METHOD FB_init : BOOL
VAR_INPUT
  /// if TRUE, the retain variables are initialized (warm start / cold start)
  bInitRetains : BOOL; 
  /// if TRUE, the instance afterwards gets moved into the copy code (online change)
  bInCopyCode  : BOOL;  
END_VAR
                  MyType := 'MC_MoveDirectOffsetFB';

ExecMode     := ExecutionMode.SEQUENCE_PRIMARY;
Priority     := PriorityLevel.NORMAL;
AbortingMode := AbortingModeEnum.BUFFER;  
SequenceFlag := SequenceFlagEnum.PRIMARY_SEQUENCE;  

                
END_METHOD

METHOD PROTECTED OnApplyOutCmd
VAR_INPUT
  /// Command message state
  State : CmdMessageState;
END_VAR
                  IF ( State = CmdMessageState.EMPTY ) 
THEN
  // Reset command outputs
  SysDepMemSet(pDest := ADR(OutCmd), Value := 0, DataLen := SIZEOF(OutCmd));         
END_IF

IF (( State = CmdMessageState.ACTIVE ) OR
    ( State = CmdMessageState.DONE   ))
THEN
  // Update results
  OutCmd.Progress          :=  PERCENT_UINT_TO_REAL( Value := _response.Progress, IsOptional := TRUE);
  OutCmd.FollowID          := _response.OriginID;
  OutCmd.RemainingDistance := _response.RemainingDistance;
END_IF
                
END_METHOD

METHOD PROTECTED OnExecRun : DINT
VAR_IN_OUT
  /// Robot assignment of function
  AxesGroup : AxesGroup; 
END_VAR
                  // call base implementation
SUPER^.OnExecRun(AxesGroup := AxesGroup);

CASE _stepCmd OF
  
  00:  IF ( _execute_R.Q ) AND ( NOT Error)  
       THEN
         // Check function is supported and parameter are valid ?
         IF (( CheckFunctionSupported( AxesGroup := AxesGroup )) AND
             ( CheckParameterValid   ( AxesGroup := AxesGroup )))      
         THEN
           // set busy flag
           Busy := TRUE;
           // Reset command outputs
           SysDepMemSet(pDest := ADR(OutCmd), Value := 0, DataLen := SIZEOF(OutCmd));         
           // apply command parameter
          _parCmd := ParCmd;
           // init parameter sequence
          _command.ParSeq := 1;
           // create command data
           CommandData := CreateCommandPayload(AxesGroup := AxesGroup);
           // Add command to active command register
          _uniqueID := AxesGroup.Acyclic.ActiveCommandRegister.AddCmd( pCommandFB := ADR(THIS^ ));     
           // set timeout
           SetTimeout(PT := _timeoutCmd, rTimer := _timerCmd);
           // inc step counter
          _stepCmd := _stepCmd + 1;
         END_IF 
       END_IF
     

  01:  // Wait for responce received
       IF ( _responseReceived )
       THEN
         // reset response received flag
        _responseReceived := FALSE;
         // update state flags
         OnUpdateStateFlags(_response.State);
         // update state flags
         OnApplyOutCmd(_response.State);
        
         // Done, Aborted or Error ?
         IF (_response.State >= CmdMessageState.DONE )
         THEN
           // set timeout
           SetTimeout(PT := _timeoutCmd, rTimer := _timerCmd);
           // inc step counter
          _stepCmd := _stepCmd + 1; 
         END_IF
       END_IF


  02: IF ( NOT Execute)
      THEN
        Reset();  
      END_IF     
ELSE
  // invalid step
  SetError( ErrorID := RobotLibraryErrorIdEnum.ERR_INVALID_STEP, Overwrite := TRUE );
END_CASE


// Reset FB
IF ( NOT Execute )
THEN
  Reset(); 
END_IF
                
END_METHOD

METHOD PROTECTED OnUpdateStateFlags
VAR_INPUT
  /// Command message state
  State : CmdMessageState;
END_VAR
                  // Reset State flags
Active             := FALSE;
CommandAborted     := FALSE;
CommandInterrupted := FALSE;
Done               := FALSE;

CASE State OF

  // No operation or process is active
  CmdMessageState.EMPTY               :;
  // Created but not yet started
  CmdMessageState.CREATED             :;
  // Buffered and awaiting execution
  CmdMessageState.BUFFERED            : CommandBuffered    := TRUE;
  // Buffered in planner for future execution
  CmdMessageState.BUFFERED_IN_PLANNER : CommandBuffered    := TRUE;
  // Currently active and in progress
  CmdMessageState.ACTIVE              : Active             := TRUE; 
  // Interrupted and awaiting continuation
  CmdMessageState.INTERRUPTED         : CommandInterrupted := TRUE;  
  // Requested for abort
  CmdMessageState.ABORT_REQUEST       :;
  // Successfully completed
  CmdMessageState.DONE                : Done               := TRUE;
                                        Busy               := FALSE;
  // Aborted before completion
  CmdMessageState.ABORTED             : CommandAborted     := TRUE;
                                        Busy               := FALSE;
  // Encountered an error during execution
  CmdMessageState.ERROR               : Error              := TRUE;
                                        Busy               := FALSE;
END_CASE
                
END_METHOD

METHOD INTERNAL ParseResponsePayload : DINT
VAR_INPUT
  /// Response data
  ResponseData : RobotLibraryResponseDataFB;
  /// Timestamp
  Timestamp    : SystemTime;  
END_VAR
VAR
  /// Parameter count
 _parameterCnt : DINT;
END_VAR
// Table 6-354: Received CMD payload (RC to PLC) of "MoveDirectOffset"
// --------------------------
// Header
// --------------------------
// Byte 00 : USINT   - ParSeq | State     
// Byte 01 : SINT    - AlarmMessageSeverity    
// Byte 02 : UINT    - AlarmMessageCode HB
// Byte 03 :         - AlarmMessageCode LB
// --------------------------
// Datablock
// --------------------------
// Byte 04 : USINT      - InvocationCounter
// Byte 05 : SINT       - Reserved
// Byte 06 : INT        - OriginID HW HB
// Byte 07 :            - OriginID HW LB
// Byte 08 : UINT       - Progress HW HB
// Byte 09 :            - Progress HW LB
// Byte 10 : REAL       - RemainingDistance HW HB
// Byte 11 :            - RemainingDistance HW LB
// Byte 12 :            - RemainingDistance LW HB
// Byte 13 :            - RemainingDistance LW LB
                  // call base implementation to parse the header from payload buffer
ResponseData.PayloadPtr := SUPER^.ParseResponsePayload(ResponseData := ResponseData, Timestamp := Timestamp);

// copy parsed header to response
_response.ParSeq               := _rspHeader.ParSeq;
_response.State                := _rspHeader.State;
_response.AlarmMessageSeverity := _rspHeader.AlarmMessageSeverity;
_response.AlarmMessageCode     := _rspHeader.AlarmMessageCode;


// Check payload remaining ? 
IF ( ResponseData.IsPayloadRemaining)
THEN
  // Get Response.InvocationCounter
 _response.InvocationCounter := ResponseData.GetUsint();
  // inc parameter counter
 _parameterCnt := _parameterCnt + 1;
END_IF

// Check payload remaining ? 
IF ( ResponseData.IsPayloadRemaining)
THEN
  // Get Response.Reserve
 _response.Reserve := ResponseData.GetSint();
  // inc parameter counter
 _parameterCnt := _parameterCnt + 1;
END_IF


// Check payload remaining ? 
IF ( ResponseData.IsPayloadRemaining)
THEN
  // Get Response.OriginID
 _response.OriginID := ResponseData.GetInt();
  // inc parameter counter
 _parameterCnt := _parameterCnt + 1;
END_IF


// Check payload remaining ? 
IF ( ResponseData.IsPayloadRemaining)
THEN
  // Get Response.Progress
 _response.Progress := ResponseData.GetUint();
  // inc parameter counter
 _parameterCnt := _parameterCnt + 1;
END_IF


// Check payload remaining ? 
IF ( ResponseData.IsPayloadRemaining)
THEN
  // Get Response.RemainingDistance
 _response.RemainingDistance := ResponseData.GetReal();
  // inc parameter counter
 _parameterCnt := _parameterCnt + 1;
END_IF
 
 
// Create logging
ParseResponsePayloadLog(ResponseData := ResponseData, Timestamp := Timestamp, ParameterCnt := _parameterCnt);
                
END_METHOD

METHOD INTERNAL ParseResponsePayloadLog
VAR_INPUT
  /// Response data
  ResponseData : RobotLibraryResponseDataFB;
  /// Timestamp
  Timestamp    : SystemTime;  
  /// Parameter count
  ParameterCnt : DINT;
END_VAR
                  // Create log entry for Parameter start
CreateLogMessagePara1 ( Timestamp   := Timestamp,
                        MessageType := MessageType.CMD,
                        Severity    := Severity.DEBUG,
                        MessageCode := 0,
                        MessageText := '{1} parameter(s) to parse from the response data:',
                        Para1       := DINT_TO_STRING(ParameterCnt));
                        

// Return if no parameter is remaining...
IF ( ParameterCnt = 0 ) THEN RETURN; END_IF
// dec remaining parameter(s)                        
ParameterCnt := ParameterCnt - 1;
// Create log entry for InvocationCounter
CreateLogMessagePara1 ( Timestamp   := Timestamp,
                        MessageType := MessageType.CMD,
                        Severity    := Severity.DEBUG,
                        MessageCode := 0,
                        MessageText := 'Response.InvocationCounter = {1}',
                        Para1       :=  USINT_TO_STRING(_response.InvocationCounter));


// Return if no parameter is remaining...
IF ( ParameterCnt = 0 ) THEN RETURN; END_IF
// dec remaining parameter(s)                        
ParameterCnt := ParameterCnt - 1;
// Create log entry for Reserve
CreateLogMessagePara1 ( Timestamp   := Timestamp,
                        MessageType := MessageType.CMD,
                        Severity    := Severity.DEBUG,
                        MessageCode := 0,
                        MessageText := 'Response.Reserve = {1}',
                        Para1       :=  SINT_TO_STRING(_response.Reserve));


// Return if no parameter is remaining...
IF ( ParameterCnt = 0 ) THEN RETURN; END_IF
// dec remaining parameter(s)                        
ParameterCnt := ParameterCnt - 1;
// Create log entry for OriginID
CreateLogMessagePara1 ( Timestamp   := Timestamp,
                        MessageType := MessageType.CMD,
                        Severity    := Severity.DEBUG,
                        MessageCode := 0,
                        MessageText := 'Response.OriginID = {1}',
                        Para1       :=  INT_TO_STRING(_response.OriginID));


// Return if no parameter is remaining...
IF ( ParameterCnt = 0 ) THEN RETURN; END_IF
// dec remaining parameter(s)                        
ParameterCnt := ParameterCnt - 1;
// Create log entry for Progress
CreateLogMessagePara1 ( Timestamp   := Timestamp,
                        MessageType := MessageType.CMD,
                        Severity    := Severity.DEBUG,
                        MessageCode := 0,
                        MessageText := 'Response.Progress = {1}',
                        Para1       :=  UINT_TO_STRING(_response.Progress));


// Return if no parameter is remaining...
IF ( ParameterCnt = 0 ) THEN RETURN; END_IF
// dec remaining parameter(s)                        
ParameterCnt := ParameterCnt - 1;
// Create log entry for RemainingDistance
CreateLogMessagePara1 ( Timestamp   := Timestamp,
                        MessageType := MessageType.CMD,
                        Severity    := Severity.DEBUG,
                        MessageCode := 0,
                        MessageText := 'Response.RemainingDistance = {1}',
                        Para1       :=  REAL_TO_STRING(_response.RemainingDistance));
                
END_METHOD

METHOD PROTECTED Reset : DINT
VAR_INPUT
END_VAR
                  Reset := SUPER^.Reset();

Done               := FALSE;
Busy               := FALSE;
Active             := FALSE;
CommandBuffered    := FALSE;
CommandAborted     := FALSE;
CommandInterrupted := FALSE;

                
END_METHOD
END_FUNCTION_BLOCK

/// Move Joints relative to relative cartesian position (Relative cartesian PTP) (Joint interpolated movement)
FUNCTION_BLOCK MC_MoveDirectRelativeFB EXTENDS RobotLibraryBaseExecuteFB
// ------------------------------------------------------------------------- 
//  SRCI Robot Library                                                
// ------------------------------------------------------------------------- 
//                                                                           
//  Object:      MoveDirectRelativeFB                                       
//  Author:      Thorsten Brach                                                
//  Date:        2024-06-01
//
//  Description:                                              
//   
//                                                                           
//  Copyright: 
//    (C) 2024 Thorsten Brach. All rights reserved                                                                                                                                            
//             Licensed under the MIT License.
//                                                                           
//  Disclaimer:                                                                           
//    This project is provided without any guarantee and can be used for   
//    private and commercial purposes. Any use is at the user’s 
//    own risk and responsibility.
//
// -------------------------------------------------------------------------
VAR_INPUT
  /// Parameter which determines the behavior towards the previously sent and still active or buffered commands
  AbortingMode       : AbortingMode;
  /// Defines the target sequence in which the command will be executed
  SequenceFlag       : SequenceFlag;
  /// command parameter
  ParCmd             : MoveDirectRelativeParCmd;       
END_VAR

VAR_OUTPUT
  /// Command is transferred and confirmed by the RC
  CommandBuffered    : BOOL;
  /// The command takes control of the motion of the according axis group
  Active             : BOOL;
  /// The command was aborted by another command.
  CommandAborted     : BOOL;
  /// TRUE, while command is interrupted during execution and can be continued
  CommandInterrupted : BOOL;
  /// command outputs
  OutCmd             : MoveDirectRelativeOutCmd;       
END_VAR



VAR
  /// internal copy of command parameter 
 _parCmd             : MoveDirectRelativeParCmd;
  /// command data to send
 _command            : MoveDirectRelativeSendData;
  /// response data received
 _response           : MoveDirectRelativeRecvData;      
END_VAR

            SUPER^(AxesGroup := AxesGroup);
          

METHOD INTERNAL CheckAddParameter : BOOL
VAR_INPUT
  /// Payload pointer
  PayloadPtr : UDINT;
END_VAR
VAR
  /// Payload as byte array
  Payload    : ARRAY [1..SIZEOF(_command)] OF BYTE;
  /// Null Byte array 
  Null       : ARRAY [1..SIZEOF(_command)] OF BYTE;
  /// Data length to compare
  DataLen    : UDINT;
END_VAR
                  // Payload pointer must be decreased by one byte, because ADR(Payload) is already one byte !
PayloadPtr := LIMIT (0, PayloadPtr - 1, SIZEOF(Payload) -1);
// Convert command struct to payload array
SysDepMemCpy( pDest := ADR(Payload), pSrc := ADR(_command), DataLen := SIZEOF(_command));
// Calculate the data length to compare - at least one byte must be compared !
DataLen := LIMIT(1, SIZEOF(Payload) - PayloadPtr, SIZEOF(Payload)); 
// Compare Payload-Array with Null-Byte-Array
CheckAddParameter := SysDepMemCmp( pData1 := ADR(Payload) + PayloadPtr , pData2 := ADR(Null), DataLen := DataLen) <>  RobotLibraryConstants.OK ;
                
END_METHOD

METHOD PROTECTED CheckFunctionSupported : BOOL
VAR_IN_OUT
  /// Robot assignment of function
  AxesGroup : AxesGroup; 
END_VAR
                  CheckFunctionSupported := AxesGroup.State.RobotData.RCSupportedFunctions.MoveDirectRelative;

IF ( NOT CheckFunctionSupported )
THEN
  // call base implementation for set error and create log entry
  SUPER^.CheckFunctionSupported(AxesGroup := AxesGroup);
END_IF
                
END_METHOD

METHOD PROTECTED CheckParameterChanged : BOOL
VAR_IN_OUT
  /// Robot assignment of function
  AxesGroup    : AxesGroup; 
END_VAR
                  // Check ParCmd Size is > 0, because MemCmp does not work correctly with size = 0
IF (SIZEOF(ParCmd) = 0) OR (_stepCmd = 0)
THEN 
  RETURN;
END_IF

// compare memory 
_parameterChanged := ( SysDepMemCmp(pData1 := ADR(ParCmd), pData2 := ADR(_parCmd), DataLen := SIZEOF(ParCmd)) <> RobotLibraryConstants.OK );

// check parameter valid ?
_parameterValid   := CheckParameterValid( AxesGroup := AxesGroup );

IF ((  _parameterChanged        )  AND 
    (  _parameterValid          )) OR
    (  _parameterUpdateInternal )  
THEN  
  // Create log entry for parameter changed event
  CreateLogMessagePara1 ( Timestamp   := AxesGroup.State.SystemTime,
                          MessageType := MessageType.CMD,
                          Severity    := Severity.DEBUG,
                          MessageCode := 0,
                          MessageText := 'NotifyParameterChanged Event {1}',
                          Para1       :=  '' );

  // reset internal flag for send parameter update
 _parameterUpdateInternal := FALSE;
  // update internal copy of parameters 
 _parCmd := ParCmd;
  // inc parameter sequence
 _command.ParSeq := _command.ParSeq + 1;
  // update command data  
  CommandData := CreateCommandPayload(AxesGroup := AxesGroup); // ( Access via reference to rCommandFB in ACR )
  // notify active command register 
  AxesGroup.Acyclic.ActiveCommandRegister.NotifyParameterChanged := _uniqueID;
END_IF
                
END_METHOD

METHOD PROTECTED CheckParameterValid : BOOL
VAR_IN_OUT
  /// Robot assignment of function
  AxesGroup : AxesGroup; 
END_VAR
VAR
  /// internal index for loops
 _idx : DINT;
END_VAR
                  CheckParameterValid := TRUE;

// Check AbortingMode valid ? 
IF (( AbortingMode <> AbortingModeEnum.BUFFER ) AND
    ( AbortingMode <> AbortingModeEnum.ABORT  ))  
THEN
  // Parameter not valid
  CheckParameterValid := FALSE;
  // Set error
  SetError( ErrorID := RobotLibraryErrorIdEnum.ERR_ABORTINGMODE_INVALID, Overwrite := TRUE );
  // Create log entry
  CreateLogMessagePara1 ( Timestamp   := AxesGroup.State.SystemTime,
                          MessageType := MessageType.CMD,
                          Severity    := Severity.ERROR,
                          MessageCode := ErrorID,
                          MessageText := 'Invalid Parameter AbortingMode = {1}',
                          Para1       := ABORTING_MODE_TO_STRING(AbortingMode));
  RETURN;                          
END_IF


// Check SequenceFlag valid ? 
IF (( SequenceFlag <> SequenceFlagEnum.PRIMARY_SEQUENCE   ) AND
    ( SequenceFlag <> SequenceFlagEnum.SECONDARY_SEQUENCE ))
THEN
  // Parameter not valid
  CheckParameterValid := FALSE;
  // Set error
  SetError( ErrorID := RobotLibraryErrorIdEnum.ERR_SEQFLAG_NOT_ALLOWED, Overwrite := TRUE );
  // Create log entry
  CreateLogMessagePara1 ( Timestamp   := AxesGroup.State.SystemTime,
                          MessageType := MessageType.CMD,
                          Severity    := Severity.ERROR,
                          MessageCode := ErrorID,
                          MessageText := 'Invalid Parameter SequenceFlag = {1}',
                          Para1       := SEQUENCE_FLAG_TO_STRING(SequenceFlag));
  RETURN;                          
END_IF


// Check ParCmd.Distance.X valid ? 
IF ( SysDepIsValidReal(ParCmd.Distance.X) = FALSE ) 
THEN
  // Parameter not valid
  CheckParameterValid := FALSE;
  // Set error
  SetError( ErrorID := RobotLibraryErrorIdEnum.ERR_INVALID_PAR_CMD, Overwrite := TRUE );
  
  // Create log entry
  CreateLogMessagePara1 ( Timestamp   := AxesGroup.State.SystemTime,
                          MessageType := MessageType.CMD,
                          Severity    := Severity.ERROR,
                          MessageCode := ErrorID,
                          MessageText := 'Invalid Parameter ParCmd.Distance.X = {1}',
                          Para1       := VALID_REAL_TO_STRING(ParCmd.Distance.X));
  RETURN;                          
END_IF


// Check ParCmd.Distance.Y valid ? 
IF ( SysDepIsValidReal(ParCmd.Distance.Y) = FALSE ) 
THEN
  // Parameter not valid
  CheckParameterValid := FALSE;
  // Set error
  SetError( ErrorID := RobotLibraryErrorIdEnum.ERR_INVALID_PAR_CMD, Overwrite := TRUE );
  
  // Create log entry
  CreateLogMessagePara1 ( Timestamp   := AxesGroup.State.SystemTime,
                          MessageType := MessageType.CMD,
                          Severity    := Severity.ERROR,
                          MessageCode := ErrorID,
                          MessageText := 'Invalid Parameter ParCmd.Distance.Y = {1}',
                          Para1       := VALID_REAL_TO_STRING(ParCmd.Distance.Y));
  RETURN;                          
END_IF


// Check ParCmd.Distance.Z valid ? 
IF ( SysDepIsValidReal(ParCmd.Distance.Z) = FALSE ) 
THEN
  // Parameter not valid
  CheckParameterValid := FALSE;
  // Set error
  SetError( ErrorID := RobotLibraryErrorIdEnum.ERR_INVALID_PAR_CMD, Overwrite := TRUE );
  
  // Create log entry
  CreateLogMessagePara1 ( Timestamp   := AxesGroup.State.SystemTime,
                          MessageType := MessageType.CMD,
                          Severity    := Severity.ERROR,
                          MessageCode := ErrorID,
                          MessageText := 'Invalid Parameter ParCmd.Distance.Z = {1}',
                          Para1       := VALID_REAL_TO_STRING(ParCmd.Distance.Z));
  RETURN;                          
END_IF


// Check ParCmd.Distance.Rx valid ? 
IF ( SysDepIsValidReal(ParCmd.Distance.Rx) = FALSE ) 
THEN
  // Parameter not valid
  CheckParameterValid := FALSE;
  // Set error
  SetError( ErrorID := RobotLibraryErrorIdEnum.ERR_INVALID_PAR_CMD, Overwrite := TRUE );
  
  // Create log entry
  CreateLogMessagePara1 ( Timestamp   := AxesGroup.State.SystemTime,
                          MessageType := MessageType.CMD,
                          Severity    := Severity.ERROR,
                          MessageCode := ErrorID,
                          MessageText := 'Invalid Parameter ParCmd.Distance.Rx = {1}',
                          Para1       := VALID_REAL_TO_STRING(ParCmd.Distance.Rx));
  RETURN;                          
END_IF


// Check ParCmd.Distance.Ry valid ? 
IF ( SysDepIsValidReal(ParCmd.Distance.Ry) = FALSE ) 
THEN
  // Parameter not valid
  CheckParameterValid := FALSE;
  // Set error
  SetError( ErrorID := RobotLibraryErrorIdEnum.ERR_INVALID_PAR_CMD, Overwrite := TRUE );
  
  // Create log entry
  CreateLogMessagePara1 ( Timestamp   := AxesGroup.State.SystemTime,
                          MessageType := MessageType.CMD,
                          Severity    := Severity.ERROR,
                          MessageCode := ErrorID,
                          MessageText := 'Invalid Parameter ParCmd.Distance.Ry = {1}',
                          Para1       := VALID_REAL_TO_STRING(ParCmd.Distance.Ry));
  RETURN;                          
END_IF


// Check ParCmd.Distance.Rz valid ? 
IF ( SysDepIsValidReal(ParCmd.Distance.Rz) = FALSE ) 
THEN
  // Parameter not valid
  CheckParameterValid := FALSE;
  // Set error
  SetError( ErrorID := RobotLibraryErrorIdEnum.ERR_INVALID_PAR_CMD, Overwrite := TRUE );
  
  // Create log entry
  CreateLogMessagePara1 ( Timestamp   := AxesGroup.State.SystemTime,
                          MessageType := MessageType.CMD,
                          Severity    := Severity.ERROR,
                          MessageCode := ErrorID,
                          MessageText := 'Invalid Parameter ParCmd.Distance.Rz = {1}',
                          Para1       := VALID_REAL_TO_STRING(ParCmd.Distance.Rz));
  RETURN;                          
END_IF


// Check ParCmd.Distance.E1 valid ? 
IF ( SysDepIsValidReal(ParCmd.Distance.E1) = FALSE ) 
THEN
  // Parameter not valid
  CheckParameterValid := FALSE;
  // Set error
  SetError( ErrorID := RobotLibraryErrorIdEnum.ERR_INVALID_PAR_CMD, Overwrite := TRUE );
  
  // Create log entry
  CreateLogMessagePara1 ( Timestamp   := AxesGroup.State.SystemTime,
                          MessageType := MessageType.CMD,
                          Severity    := Severity.ERROR,
                          MessageCode := ErrorID,
                          MessageText := 'Invalid Parameter ParCmd.Distance.E1 = {1}',
                          Para1       := VALID_REAL_TO_STRING(ParCmd.Distance.E1));
  RETURN;                          
END_IF


// Check ParCmd.Distance.E2 valid ? 
IF ( SysDepIsValidReal(ParCmd.Distance.E2) = FALSE ) 
THEN
  // Parameter not valid
  CheckParameterValid := FALSE;
  // Set error
  SetError( ErrorID := RobotLibraryErrorIdEnum.ERR_INVALID_PAR_CMD, Overwrite := TRUE );
  
  // Create log entry
  CreateLogMessagePara1 ( Timestamp   := AxesGroup.State.SystemTime,
                          MessageType := MessageType.CMD,
                          Severity    := Severity.ERROR,
                          MessageCode := ErrorID,
                          MessageText := 'Invalid Parameter ParCmd.Distance.E2 = {1}',
                          Para1       := VALID_REAL_TO_STRING(ParCmd.Distance.E2));
  RETURN;                          
END_IF


// Check ParCmd.Distance.E3 valid ? 
IF ( SysDepIsValidReal(ParCmd.Distance.E3) = FALSE ) 
THEN
  // Parameter not valid
  CheckParameterValid := FALSE;
  // Set error
  SetError( ErrorID := RobotLibraryErrorIdEnum.ERR_INVALID_PAR_CMD, Overwrite := TRUE );
  
  // Create log entry
  CreateLogMessagePara1 ( Timestamp   := AxesGroup.State.SystemTime,
                          MessageType := MessageType.CMD,
                          Severity    := Severity.ERROR,
                          MessageCode := ErrorID,
                          MessageText := 'Invalid Parameter ParCmd.Distance.E3 = {1}',
                          Para1       := VALID_REAL_TO_STRING(ParCmd.Distance.E3));
  RETURN;                          
END_IF


// Check ParCmd.Distance.E4 valid ? 
IF ( SysDepIsValidReal(ParCmd.Distance.E4) = FALSE ) 
THEN
  // Parameter not valid
  CheckParameterValid := FALSE;
  // Set error
  SetError( ErrorID := RobotLibraryErrorIdEnum.ERR_INVALID_PAR_CMD, Overwrite := TRUE );
  
  // Create log entry
  CreateLogMessagePara1 ( Timestamp   := AxesGroup.State.SystemTime,
                          MessageType := MessageType.CMD,
                          Severity    := Severity.ERROR,
                          MessageCode := ErrorID,
                          MessageText := 'Invalid Parameter ParCmd.Distance.E4 = {1}',
                          Para1       := VALID_REAL_TO_STRING(ParCmd.Distance.E4));
  RETURN;                          
END_IF


// Check ParCmd.Distance.E5 valid ? 
IF ( SysDepIsValidReal(ParCmd.Distance.E5) = FALSE ) 
THEN
  // Parameter not valid
  CheckParameterValid := FALSE;
  // Set error
  SetError( ErrorID := RobotLibraryErrorIdEnum.ERR_INVALID_PAR_CMD, Overwrite := TRUE );
  
  // Create log entry
  CreateLogMessagePara1 ( Timestamp   := AxesGroup.State.SystemTime,
                          MessageType := MessageType.CMD,
                          Severity    := Severity.ERROR,
                          MessageCode := ErrorID,
                          MessageText := 'Invalid Parameter ParCmd.Distance.E5 = {1}',
                          Para1       := VALID_REAL_TO_STRING(ParCmd.Distance.E5));
  RETURN;                          
END_IF


// Check ParCmd.Distance.E6 valid ? 
IF ( SysDepIsValidReal(ParCmd.Distance.E6) = FALSE ) 
THEN
  // Parameter not valid
  CheckParameterValid := FALSE;
  // Set error
  SetError( ErrorID := RobotLibraryErrorIdEnum.ERR_INVALID_PAR_CMD, Overwrite := TRUE );
  
  // Create log entry
  CreateLogMessagePara1 ( Timestamp   := AxesGroup.State.SystemTime,
                          MessageType := MessageType.CMD,
                          Severity    := Severity.ERROR,
                          MessageCode := ErrorID,
                          MessageText := 'Invalid Parameter ParCmd.Distance.E6 = {1}',
                          Para1       := VALID_REAL_TO_STRING(ParCmd.Distance.E6));
  RETURN;                          
END_IF


// Check ParCmd.Distance.Config.Shoulder valid ? 
IF (( ParCmd.Distance.Config.Shoulder <> ArmConfigShoulder.USE_CONFIG ) AND  
    ( ParCmd.Distance.Config.Shoulder <> ArmConfigShoulder.SAME       ) AND
    ( ParCmd.Distance.Config.Shoulder <> ArmConfigShoulder.FREE       ) AND
    ( ParCmd.Distance.Config.Shoulder <> ArmConfigShoulder.BACK       ) AND
    ( ParCmd.Distance.Config.Shoulder <> ArmConfigShoulder.FRONT      ))
THEN
  // Parameter not valid
  CheckParameterValid := FALSE;
  // Set error
  SetError( ErrorID := RobotLibraryErrorIdEnum.ERR_CONFIGMODE_SHOULDER_INVALID, Overwrite := TRUE );
  // Create log entry
  CreateLogMessagePara1 ( Timestamp   := AxesGroup.State.SystemTime,
                          MessageType := MessageType.CMD,
                          Severity    := Severity.ERROR,
                          MessageCode := ErrorID,
                          MessageText := 'Invalid Parameter ParCmd.Distance.Config.Shoulder = {1}',
                          Para1       :=  ARM_CONFIG_SHOULDER_TO_STRING(ParCmd.Distance.Config.Shoulder));
  RETURN;                          
END_IF


// Check ParCmd.Distance.Config.Elbow valid ? 
IF (( ParCmd.Distance.Config.Elbow <> ArmConfigElbow.USE_CONFIG ) AND  
    ( ParCmd.Distance.Config.Elbow <> ArmConfigElbow.SAME       ) AND
    ( ParCmd.Distance.Config.Elbow <> ArmConfigElbow.FREE       ) AND
    ( ParCmd.Distance.Config.Elbow <> ArmConfigElbow.DOWN       ) AND
    ( ParCmd.Distance.Config.Elbow <> ArmConfigElbow.UP         ))
THEN
  // Parameter not valid
  CheckParameterValid := FALSE;
  // Set error
  SetError( ErrorID := RobotLibraryErrorIdEnum.ERR_CONFIGMODE_ELBOW_INVALID, Overwrite := TRUE );
  // Create log entry
  CreateLogMessagePara1 ( Timestamp   := AxesGroup.State.SystemTime,
                          MessageType := MessageType.CMD,
                          Severity    := Severity.ERROR,
                          MessageCode := ErrorID,
                          MessageText := 'Invalid Parameter ParCmd.Distance.Config.Elbow = {1}',
                          Para1       :=  ARM_CONFIG_ELBOW_TO_STRING(ParCmd.Distance.Config.Elbow));
  RETURN;                          
END_IF


// Check ParCmd.Distance.Config.Wrist valid ? 
IF (( ParCmd.Distance.Config.Wrist <> ArmConfigWrist.USE_CONFIG ) AND  
    ( ParCmd.Distance.Config.Wrist <> ArmConfigWrist.SAME       ) AND
    ( ParCmd.Distance.Config.Wrist <> ArmConfigWrist.FREE       ) AND
    ( ParCmd.Distance.Config.Wrist <> ArmConfigWrist.FLIP       ) AND
    ( ParCmd.Distance.Config.Wrist <> ArmConfigWrist.NON_FLIP   ))
THEN
  // Parameter not valid
  CheckParameterValid := FALSE;
  // Set error
  SetError( ErrorID := RobotLibraryErrorIdEnum.ERR_CONFIGMODE_WRIST_INVALID, Overwrite := TRUE );
  // Create log entry
  CreateLogMessagePara1 ( Timestamp   := AxesGroup.State.SystemTime,
                          MessageType := MessageType.CMD,
                          Severity    := Severity.ERROR,
                          MessageCode := ErrorID,
                          MessageText := 'Invalid Parameter ParCmd.Distance.Config.Wrist = {1}',
                          Para1       :=  ARM_CONFIG_WRIST_TO_STRING(ParCmd.Distance.Config.Wrist));
  RETURN;                          
END_IF


// Check ParCmd.ReferenceType valid ? 
IF (( ParCmd.ReferenceType <> ReferenceType.TOOL  ) AND
    ( ParCmd.ReferenceType <> ReferenceType.FRAME ))  
THEN
  // Parameter not valid
  CheckParameterValid := FALSE;
  // Set error
  SetError( ErrorID := RobotLibraryErrorIdEnum.ERR_INVALID_PAR_CMD, Overwrite := TRUE );
  // Create log entry
  CreateLogMessagePara1 ( Timestamp   := AxesGroup.State.SystemTime,
                          MessageType := MessageType.CMD,
                          Severity    := Severity.ERROR,
                          MessageCode := ErrorID,
                          MessageText := 'Invalid Parameter ParCmd.ReferenceType = {1}',
                          Para1       := REFERENCE_TYPE_TO_STRING(ParCmd.ReferenceType));
  RETURN;                          
END_IF


// Check ParCmd.VelocityRate valid ? 
IF  (( SysDepIsValidReal(ParCmd.VelocityRate) = FALSE )  OR
    ((                   ParCmd.VelocityRate  <     0 )  AND 
     (                   ParCmd.VelocityRate <>    -1 )) OR   
     (                   ParCmd.VelocityRate  >   100 ))      
THEN
  // Parameter not valid
  CheckParameterValid := FALSE;
  // Set error
  SetError( ErrorID := RobotLibraryErrorIdEnum.ERR_VELOCITY_INVALID, Overwrite := TRUE );
  // Create log entry
  CreateLogMessagePara1 ( Timestamp   := AxesGroup.State.SystemTime,
                          MessageType := MessageType.CMD,
                          Severity    := Severity.ERROR,
                          MessageCode := ErrorID,
                          MessageText := 'Invalid Parameter ParCmd.VelocityRate = {1}',
                          Para1       := VALID_REAL_TO_STRING(ParCmd.VelocityRate));                            
  RETURN;
END_IF


// Check ParCmd.AccelerationRate valid ? 
IF  (( SysDepIsValidReal(ParCmd.AccelerationRate) = FALSE )  OR
    ((                   ParCmd.AccelerationRate  <     0 )  AND 
     (                   ParCmd.AccelerationRate <>    -1 )) OR   
     (                   ParCmd.AccelerationRate  >   100 ))      
THEN
  // Parameter not valid
  CheckParameterValid := FALSE;
  // Set error
  SetError( ErrorID := RobotLibraryErrorIdEnum.ERR_ACCELERATION_INVALID, Overwrite := TRUE );
  // Create log entry
  CreateLogMessagePara1 ( Timestamp   := AxesGroup.State.SystemTime,
                          MessageType := MessageType.CMD,
                          Severity    := Severity.ERROR,
                          MessageCode := ErrorID,
                          MessageText := 'Invalid Parameter ParCmd.AccelerationRate = {1}',
                          Para1       := VALID_REAL_TO_STRING(ParCmd.AccelerationRate));                            
  RETURN;
END_IF


// Check ParCmd.DecelerationRate valid ? 
IF  (( SysDepIsValidReal(ParCmd.DecelerationRate) = FALSE )  OR
    ((                   ParCmd.DecelerationRate  <     0 )  AND 
     (                   ParCmd.DecelerationRate <>    -1 )) OR   
     (                   ParCmd.DecelerationRate  >   100 ))      
THEN
  // Parameter not valid
  CheckParameterValid := FALSE;
  // Set error
  SetError( ErrorID := RobotLibraryErrorIdEnum.ERR_DECELERATION_INVALID, Overwrite := TRUE );
  // Create log entry
  CreateLogMessagePara1 ( Timestamp   := AxesGroup.State.SystemTime,
                          MessageType := MessageType.CMD,
                          Severity    := Severity.ERROR,
                          MessageCode := ErrorID,
                          MessageText := 'Invalid Parameter ParCmd.DecelerationRate = {1}',
                          Para1       := VALID_REAL_TO_STRING(ParCmd.DecelerationRate));                            
  RETURN;
END_IF


// Check ParCmd.JerkRate valid ? 
IF  (( SysDepIsValidReal(ParCmd.JerkRate) = FALSE )  OR
    ((                   ParCmd.JerkRate  <     0 )  AND 
     (                   ParCmd.JerkRate <>    -1 )) OR   
     (                   ParCmd.JerkRate  >   100 ))      
THEN
  // Parameter not valid
  CheckParameterValid := FALSE;
  // Set error
  SetError( ErrorID := RobotLibraryErrorIdEnum.ERR_JERK_INVALID, Overwrite := TRUE );
  // Create log entry
  CreateLogMessagePara1 ( Timestamp   := AxesGroup.State.SystemTime,
                          MessageType := MessageType.CMD,
                          Severity    := Severity.ERROR,
                          MessageCode := ErrorID,
                          MessageText := 'Invalid Parameter ParCmd.JerkRate = {1}',
                          Para1       := VALID_REAL_TO_STRING(ParCmd.JerkRate));                            
  RETURN;
END_IF


// Check ParCmd.ToolNo valid ? 
IF (( ParCmd.ToolNo <   0                                                ) OR   
    ( ParCmd.ToolNo > 254                                                ) OR
    ( ParCmd.ToolNo > AxesGroup.State.ConfigurationData.HighestToolIndex ) OR
    ( ParCmd.ToolNo > AxesGroup.State.UnifiedToolIndex                   ))    
THEN
  // Parameter not valid
  CheckParameterValid := FALSE;
  
  // Check ToolNo available on RC ? 
  IF ( ParCmd.ToolNo > AxesGroup.State.ConfigurationData.HighestToolIndex )
  THEN
    SetError( ErrorID := RobotLibraryErrorIdEnum.ERR_TOOLNO_UNAVAILABLE, Overwrite := TRUE );
  ELSE
    SetError( ErrorID := RobotLibraryErrorIdEnum.ERR_TOOLNO_RANGE, Overwrite := TRUE );
	END_IF  
  
  // Create log entry
  CreateLogMessagePara1 ( Timestamp   := AxesGroup.State.SystemTime,
                          MessageType := MessageType.CMD,
                          Severity    := Severity.ERROR,
                          MessageCode := ErrorID,
                          MessageText := 'Invalid Parameter ParCmd.ToolNo = {1}',
                          Para1       := USINT_TO_STRING(ParCmd.ToolNo));                            
  RETURN;
END_IF


// Check ParCmd.FrameNo valid ? 
IF (( ParCmd.FrameNo <   0                                                 ) OR   
    ( ParCmd.FrameNo > 254                                                 ) OR
    ( ParCmd.FrameNo > AxesGroup.State.ConfigurationData.HighestFrameIndex ) OR
    ( ParCmd.FrameNo > AxesGroup.State.UnifiedFrameIndex                   ))         
THEN
  // Parameter not valid
  CheckParameterValid := FALSE;
  
  // Check FrameNo available on RC ? 
  IF ( ParCmd.FrameNo > AxesGroup.State.ConfigurationData.HighestFrameIndex )
  THEN
    SetError( ErrorID := RobotLibraryErrorIdEnum.ERR_FRAMENO_UNAVAILABLE, Overwrite := TRUE );
  ELSE
    SetError( ErrorID := RobotLibraryErrorIdEnum.ERR_FRAMENO_RANGE, Overwrite := TRUE );
	END_IF  
  
  // Create log entry
  CreateLogMessagePara1 ( Timestamp   := AxesGroup.State.SystemTime,
                          MessageType := MessageType.CMD,
                          Severity    := Severity.ERROR,
                          MessageCode := ErrorID,
                          MessageText := 'Invalid Parameter ParCmd.FrameNo = {1}',
                          Para1       := USINT_TO_STRING(ParCmd.FrameNo));                            
  RETURN;
END_IF


// Check ParCmd.BlendingMode valid ? 
IF (( ParCmd.BlendingMode <> BlendingMode.EXACT_STOP           ) AND   
    ( ParCmd.BlendingMode <> BlendingMode.DEFINED_VELOCITY     ) AND
    ( ParCmd.BlendingMode <> BlendingMode.CORNER_DISTANCE      ) AND
    ( ParCmd.BlendingMode <> BlendingMode.MAX_CORNER_DEVIATION ) AND
    ( ParCmd.BlendingMode <> BlendingMode.CORNER_DISTANCE_2R   ) AND
    ( ParCmd.BlendingMode <> BlendingMode.RAMP_OVERLAP         ) AND
    ( ParCmd.BlendingMode <> BlendingMode.CORNER_DISTANCE_1R   ))    
THEN
  // Parameter not valid
  CheckParameterValid := FALSE;
  // Set error
  SetError( ErrorID := RobotLibraryErrorIdEnum.ERR_INVALID_PAR_CMD, Overwrite := TRUE );
  // Create log entry
  CreateLogMessagePara1 ( Timestamp   := AxesGroup.State.SystemTime,
                          MessageType := MessageType.CMD,
                          Severity    := Severity.ERROR,
                          MessageCode := ErrorID,
                          MessageText := 'Invalid Parameter ParCmd.BlendingMode = {1}',
                          Para1       := BLENDING_MODE_TO_STRING(ParCmd.BlendingMode));                            
  RETURN;
END_IF


FOR _idx := 0 TO 1 
DO
  // Check ParCmd.BlendingParameter valid ? 
  IF  ( SysDepIsValidReal(ParCmd.BlendingParameter[_idx]) = FALSE ) 
  THEN
    // Parameter not valid
    CheckParameterValid := FALSE;
    // Set error
    SetError( ErrorID := RobotLibraryErrorIdEnum.ERR_JERK_INVALID, Overwrite := TRUE );
    // Create log entry
    CreateLogMessagePara2 ( Timestamp   := AxesGroup.State.SystemTime,
                            MessageType := MessageType.CMD,
                            Severity    := Severity.ERROR,
                            MessageCode := ErrorID,
                            MessageText := 'Invalid Parameter ParCmd.BlendingParameter[{2}] = {1}',
                            Para1       := VALID_REAL_TO_STRING(ParCmd.JerkRate),
                            Para2       := DINT_TO_STRING(_idx));       
    EXIT;                     
    RETURN;
  END_IF
END_FOR


// Check ParCmd.MoveTime valid ? 
IF  ( ParCmd.MoveTime < T#0S )
THEN
  // Parameter not valid
  CheckParameterValid := FALSE;
  // Set error
  SetError( ErrorID := RobotLibraryErrorIdEnum.ERR_INVALID_PAR_CMD, Overwrite := TRUE );
  // Create log entry
  CreateLogMessagePara1 ( Timestamp   := AxesGroup.State.SystemTime,
                          MessageType := MessageType.CMD,
                          Severity    := Severity.ERROR,
                          MessageCode := ErrorID,
                          MessageText := 'Invalid Parameter ParCmd.MoveTime = {1}',
                          Para1       := TIME_TO_STRING(ParCmd.MoveTime));                            
  RETURN;
END_IF


// Check ParCmd.ConfigMode.Shoulder valid ? 
IF (( ParCmd.ConfigMode.Shoulder <> ArmConfigShoulder.USE_CONFIG ) AND  
    ( ParCmd.ConfigMode.Shoulder <> ArmConfigShoulder.SAME       ) AND
    ( ParCmd.ConfigMode.Shoulder <> ArmConfigShoulder.FREE       ) AND
    ( ParCmd.ConfigMode.Shoulder <> ArmConfigShoulder.BACK       ) AND
    ( ParCmd.ConfigMode.Shoulder <> ArmConfigShoulder.FRONT      ))
THEN
  // Parameter not valid
  CheckParameterValid := FALSE;
  // Set error
  SetError( ErrorID := RobotLibraryErrorIdEnum.ERR_INVALID_PAR_CMD, Overwrite := TRUE );
  // Create log entry
  CreateLogMessagePara1 ( Timestamp   := AxesGroup.State.SystemTime,
                          MessageType := MessageType.CMD,
                          Severity    := Severity.ERROR,
                          MessageCode := ErrorID,
                          MessageText := 'Invalid Parameter ParCmd.ConfigMode.Shoulder = {1}',
                          Para1       :=  ARM_CONFIG_SHOULDER_TO_STRING(ParCmd.ConfigMode.Shoulder));
  RETURN;                          
END_IF


// Check ParCmd.ConfigMode.Elbow valid ? 
IF (( ParCmd.ConfigMode.Elbow <> ArmConfigElbow.USE_CONFIG ) AND  
    ( ParCmd.ConfigMode.Elbow <> ArmConfigElbow.SAME       ) AND
    ( ParCmd.ConfigMode.Elbow <> ArmConfigElbow.FREE       ) AND
    ( ParCmd.ConfigMode.Elbow <> ArmConfigElbow.DOWN       ) AND
    ( ParCmd.ConfigMode.Elbow <> ArmConfigElbow.UP         ))
THEN
  // Parameter not valid
  CheckParameterValid := FALSE;
  // Set error
  SetError( ErrorID := RobotLibraryErrorIdEnum.ERR_INVALID_PAR_CMD, Overwrite := TRUE );
  // Create log entry
  CreateLogMessagePara1 ( Timestamp   := AxesGroup.State.SystemTime,
                          MessageType := MessageType.CMD,
                          Severity    := Severity.ERROR,
                          MessageCode := ErrorID,
                          MessageText := 'Invalid Parameter ParCmd.ConfigMode.Elbow = {1}',
                          Para1       :=  ARM_CONFIG_ELBOW_TO_STRING(ParCmd.ConfigMode.Elbow));
  RETURN;                          
END_IF


// Check ParCmd.ConfigMode.Wrist valid ? 
IF (( ParCmd.ConfigMode.Wrist <> ArmConfigWrist.USE_CONFIG ) AND  
    ( ParCmd.ConfigMode.Wrist <> ArmConfigWrist.SAME       ) AND
    ( ParCmd.ConfigMode.Wrist <> ArmConfigWrist.FREE       ) AND
    ( ParCmd.ConfigMode.Wrist <> ArmConfigWrist.FLIP       ) AND
    ( ParCmd.ConfigMode.Wrist <> ArmConfigWrist.NON_FLIP   ))
THEN
  // Parameter not valid
  CheckParameterValid := FALSE;
  // Set error
  SetError( ErrorID := RobotLibraryErrorIdEnum.ERR_INVALID_PAR_CMD, Overwrite := TRUE );
  // Create log entry
  CreateLogMessagePara1 ( Timestamp   := AxesGroup.State.SystemTime,
                          MessageType := MessageType.CMD,
                          Severity    := Severity.ERROR,
                          MessageCode := ErrorID,
                          MessageText := 'Invalid Parameter ParCmd.ConfigMode.Wrist = {1}',
                          Para1       :=  ARM_CONFIG_WRIST_TO_STRING(ParCmd.ConfigMode.Wrist));
  RETURN;                          
END_IF


// Check ParCmd.TurnMode valid ? 
IF (( ParCmd.TurnMode <> TurnMode.USE_TURN_NUMBER ) AND  
    ( ParCmd.TurnMode <> TurnMode.SAME            ) AND
    ( ParCmd.TurnMode <> TurnMode.FREE            ))
THEN
  // Parameter not valid
  CheckParameterValid := FALSE;
  // Set error
  SetError( ErrorID := RobotLibraryErrorIdEnum.ERR_INVALID_PAR_CMD, Overwrite := TRUE );
  // Create log entry
  CreateLogMessagePara1 ( Timestamp   := AxesGroup.State.SystemTime,
                          MessageType := MessageType.CMD,
                          Severity    := Severity.ERROR,
                          MessageCode := ErrorID,
                          MessageText := 'Invalid Parameter ParCmd.TurnMode = {1}',
                          Para1       :=  TURN_MODE_TO_STRING(ParCmd.TurnMode));
  RETURN;                          
END_IF


// Check ParCmd.Manipulation
// -> no plausibility check for boolean


FOR _idx := 0 TO 3 
DO
  // Check ParCmd.EmitterID valid ? 
  IF  (( ParCmd.EmitterID[_idx] < -127 ) OR
       ( ParCmd.EmitterID[_idx] >  127 ))     
  THEN
    // Parameter not valid
    CheckParameterValid := FALSE;
    // Set error
    SetError( ErrorID := RobotLibraryErrorIdEnum.ERR_INVALID_PAR_CMD, Overwrite := TRUE );
    // Create log entry
    CreateLogMessagePara2 ( Timestamp   := AxesGroup.State.SystemTime,
                            MessageType := MessageType.CMD,
                            Severity    := Severity.ERROR,
                            MessageCode := ErrorID,
                            MessageText := 'Invalid Parameter ParCmd.EmitterID[{2}] = {1}',
                            Para1       := SINT_TO_STRING(ParCmd.EmitterID[_idx]),
                            Para2       := DINT_TO_STRING(_idx));       
    EXIT;                     
    RETURN;
  END_IF
END_FOR
                
END_METHOD

METHOD INTERNAL CreateCommandPayload : RobotLibraryCommandDataFB
VAR_IN_OUT
  /// Robot assignment of function
  AxesGroup : AxesGroup; 
END_VAR
VAR
  /// internal index for loops
 _idx          : DINT;
  /// Parameter count
 _parameterCnt : DINT;
END_VAR
// Table 6-297: Sent CMD payload (PLC to RC) of "MoveDirectRelative"
// --------------------------
// Header
// --------------------------
// Byte 00 : UINT  - Type HB     
// Byte 01 :       - Type LB    
// Byte 02 : USINT - Reserve | ExecutionMode
// Byte 03 : USINT - ParSeq  | Priority
// --------------------------
// Datablock
// --------------------------
// Byte 04 : SINT       - EmitterID[0]
// Byte 05 : SINT       - EmitterID[1]
// Byte 06 : SINT       - EmitterID[2]
// Byte 07 : SINT       - EmitterID[3]
// Byte 08 : SINT       - ListenerID
// Byte 09 : BYTE       - Reserved
// Byte 10 : UINT       - VelocityRate HW HB
// Byte 11 :            - VelocityRate HW LB
// Byte 12 : UINT       - AccelerationRate HW HB
// Byte 13 :            - AccelerationRate HW LB
// Byte 14 : UINT       - DecelerationRate HW HB
// Byte 15 :            - DecelerationRate HW LB
// Byte 16 : UINT       - JerkRate HW HB
// Byte 17 :            - JerkRate HW LB
// Byte 18 : USINT      - ToolNo
// Byte 19 : USINT      - FrameNo
// Byte 20 : USINT      - BlendingMode
// Byte 21 : Byte       - Reserve
// Byte 22 : REAL       - BlendingParameter[0] HW HB
// Byte 23 :            - BlendingParameter[0] HW LB
// Byte 24 :            - BlendingParameter[0] LW HB
// Byte 25 :            - BlendingParameter[0] LW LB
// Byte 26 : REAL       - BlendingParameter[1] HW HB
// Byte 27 :            - BlendingParameter[1] HW LB
// Byte 28 :            - BlendingParameter[1] LW HB
// Byte 29 :            - BlendingParameter[1] LW LB
// Byte 30 : REAL       - Distance.X HW HB
// Byte 31 :            - Distance.X HW LB
// Byte 32 :            - Distance.X LW HB
// Byte 33 :            - Distance.X LW LB
// Byte 34 : REAL       - Distance.Y HW HB
// Byte 35 :            - Distance.Y HW LB
// Byte 36 :            - Distance.Y LW HB
// Byte 37 :            - Distance.Y LW LB
// Byte 38 : REAL       - Distance.Z HW HB
// Byte 39 :            - Distance.Z HW LB
// Byte 40 :            - Distance.Z LW HB
// Byte 41 :            - Distance.Z LW LB
// Byte 42 : REAL       - Distance.RX HW HB
// Byte 43 :            - Distance.RX HW LB
// Byte 44 :            - Distance.RX LW HB
// Byte 45 :            - Distance.RX LW LB
// Byte 46 : REAL       - Distance.RY HW HB
// Byte 47 :            - Distance.RY HW LB
// Byte 48 :            - Distance.RY LW HB
// Byte 49 :            - Distance.RY LW LB
// Byte 50 : REAL       - Distance.RZ HW HB
// Byte 51 :            - Distance.RZ HW LB
// Byte 52 :            - Distance.RZ LW HB
// Byte 53 :            - Distance.RZ LW LB
// Byte 54 : BYTE       - - - - - W E S
// Byte 55 : BYTE       - Reserved
// Byte 56 : BYTE       - Distance.TurnNumber[0]
// Byte 57 : BYTE       - Distance.TurnNumber[1]
// Byte 58 : BYTE       - Distance.TurnNumber[2]
// Byte 59 : BYTE       - Distance.TurnNumber[3]
// Byte 60 : REAL       - Distance.E1 HW HB
// Byte 61 :            - Distance.E1 HW LB
// Byte 62 :            - Distance.E1 LW HB
// Byte 63 :            - Distance.E1 LW LB
// Byte 64 : BOOL       - Manipulation
// Byte 65 : BYTE       - Reserved
// Byte 66 : BYTE       - ConfigMode[0]
// Byte 67 : BYTE       - ConfigMode[1]
// Byte 68 : USINT      - ReferenceType
// Byte 69 : USINT      - TurnMode
// Byte 70 : UINT       - Time HW HB
// Byte 71 :            - Time HW LB
// Byte 72 : REAL       - Distance.E2 HW HB
// Byte 73 :            - Distance.E2 HW LB
// Byte 74 :            - Distance.E2 LW HB
// Byte 75 :            - Distance.E2 LW LB
// Byte 76 : REAL       - Distance.E3 HW HB
// Byte 77 :            - Distance.E3 HW LB
// Byte 78 :            - Distance.E3 LW HB
// Byte 79 :            - Distance.E3 LW LB
// Byte 80 : REAL       - Distance.E4 HW HB
// Byte 81 :            - Distance.E4 HW LB
// Byte 82 :            - Distance.E4 LW HB
// Byte 83 :            - Distance.E4 LW LB
// Byte 84 : REAL       - Distance.E5 HW HB
// Byte 85 :            - Distance.E5 HW LB
// Byte 86 :            - Distance.E5 LW HB
// Byte 87 :            - Distance.E5 LW LB
// Byte 88 : REAL       - Distance.E6 HW HB
// Byte 89 :            - Distance.E6 HW LB
// Byte 90 :            - Distance.E6 LW HB
// Byte 91 :            - Distance.E6 LW LB
// --------------------------
                  // set command parameter 
_command.CmdTyp            :=  CmdType.MoveDirectRelative;
_command.ExecMode          :=  ExecMode;
_command.ParSeq            := _command.ParSeq;
_command.Priority          :=  Priority;
_command.EmitterID         := _parCmd.EmitterID;
_command.ListenerID        := 0;
_command.Reserve           := 0;
_command.VelocityRate      := REAL_TO_PERCENT_UINT(_parCmd.VelocityRate     , IsOptional := FALSE);
_command.AccelerationRate  := REAL_TO_PERCENT_UINT(_parCmd.AccelerationRate , IsOptional := FALSE);
_command.DecelerationRate  := REAL_TO_PERCENT_UINT(_parCmd.DecelerationRate , IsOptional := TRUE );
_command.JerkRate          := REAL_TO_PERCENT_UINT(_parCmd.JerkRate         , IsOptional := TRUE );
_command.ToolNo            := _parCmd.ToolNo;
_command.FrameNo           := _parCmd.FrameNo;
_command.BlendingMode      := _parCmd.BlendingMode;
_command.Reserve2          := 0;
_command.BlendingParameter := _parCmd.BlendingParameter;
_command.Distance          := _parCmd.Distance;
_command.Manipulation      := _parCmd.Manipulation;
_command.Reserve3          := 0;
_command.ConfigMode        :=  ArmConfigParameterToBytes(_parCmd.ConfigMode);
_command.ReferenceType     := _parCmd.ReferenceType;
_command.TurnMode          := _parCmd.TurnMode;
_command.MoveTime          := TIME_TO_UINT(_parCmd.MoveTime);


// copy command data to header
_cmdHeader := _command;
// call base implementation to copy header to payload buffer
CreateCommandPayload := SUPER^.CreateCommandPayload(AxesGroup := AxesGroup);


FOR _idx := 0 TO 3 
DO
  // Check parameter must be added ? 
  IF ( CheckAddParameter(CreateCommandPayload.PayloadPtr))
  THEN
    // add command.EmitterID[x]
    CreateCommandPayload.AddSint(_command.EmitterID[_idx]);
    // inc parameter counter
   _parameterCnt := _parameterCnt + 1;  
  END_IF
END_FOR


// Check parameter must be added ? 
IF ( CheckAddParameter(CreateCommandPayload.PayloadPtr))
THEN
  // add command.ListenerID
  CreateCommandPayload.AddSint(_command.ListenerID);
  // inc parameter counter
 _parameterCnt := _parameterCnt + 1;  
END_IF


// Check parameter must be added ? 
IF ( CheckAddParameter(CreateCommandPayload.PayloadPtr))
THEN
  // add command.Reserve
  CreateCommandPayload.AddByte(_command.Reserve);
  // inc parameter counter
 _parameterCnt := _parameterCnt + 1;  
END_IF


// Check parameter must be added ? 
IF ( CheckAddParameter(CreateCommandPayload.PayloadPtr))
THEN
  // add command.VelocityRate
  CreateCommandPayload.AddUint(_command.VelocityRate);
  // inc parameter counter
 _parameterCnt := _parameterCnt + 1;  
END_IF


// Check parameter must be added ? 
IF ( CheckAddParameter(CreateCommandPayload.PayloadPtr))
THEN
  // add command.AccelerationRate
  CreateCommandPayload.AddUint(_command.AccelerationRate);
  // inc parameter counter
 _parameterCnt := _parameterCnt + 1;  
END_IF


// Check parameter must be added ? 
IF ( CheckAddParameter(CreateCommandPayload.PayloadPtr))
THEN
  // add command.DecelerationRate
  CreateCommandPayload.AddUint(_command.DecelerationRate);
  // inc parameter counter
 _parameterCnt := _parameterCnt + 1;  
END_IF


// Check parameter must be added ? 
IF ( CheckAddParameter(CreateCommandPayload.PayloadPtr))
THEN
  // add command.JerkRate
  CreateCommandPayload.AddUint(_command.JerkRate);
  // inc parameter counter
 _parameterCnt := _parameterCnt + 1;  
END_IF


// Check parameter must be added ? 
IF ( CheckAddParameter(CreateCommandPayload.PayloadPtr))
THEN
  // add command.ToolNo
  CreateCommandPayload.AddUsint(_command.ToolNo);
  // inc parameter counter
 _parameterCnt := _parameterCnt + 1;  
END_IF


// Check parameter must be added ? 
IF ( CheckAddParameter(CreateCommandPayload.PayloadPtr))
THEN
  // add command.mFrameNo
  CreateCommandPayload.AddUsint(_command.FrameNo);
  // inc parameter counter
 _parameterCnt := _parameterCnt + 1;  
END_IF


// Check parameter must be added ? 
IF ( CheckAddParameter(CreateCommandPayload.PayloadPtr))
THEN
  // add command.BlendingMode
  CreateCommandPayload.AddUsint(_command.BlendingMode);
  // inc parameter counter
 _parameterCnt := _parameterCnt + 1;  
END_IF


// Check parameter must be added ? 
IF ( CheckAddParameter(CreateCommandPayload.PayloadPtr))
THEN
  // add command.Reserve2
  CreateCommandPayload.AddByte(_command.Reserve2);
  // inc parameter counter
 _parameterCnt := _parameterCnt + 1;  
END_IF


// Check parameter must be added ? 
IF ( CheckAddParameter(CreateCommandPayload.PayloadPtr))
THEN
  // add command.BlendingParameter[0]
  CreateCommandPayload.AddReal(_command.BlendingParameter[0]);
  // inc parameter counter
 _parameterCnt := _parameterCnt + 1;  
END_IF


// Check parameter must be added ? 
IF ( CheckAddParameter(CreateCommandPayload.PayloadPtr))
THEN
  // add command.BlendingParameter[1]
  CreateCommandPayload.AddReal(_command.BlendingParameter[1]);
  // inc parameter counter
 _parameterCnt := _parameterCnt + 1;  
END_IF


// Check parameter must be added ? 
IF ( CheckAddParameter(CreateCommandPayload.PayloadPtr))
THEN
  // add command.Distance.X
  CreateCommandPayload.AddReal(_command.Distance.X);
  // inc parameter counter
 _parameterCnt := _parameterCnt + 1;  
END_IF


// Check parameter must be added ? 
IF ( CheckAddParameter(CreateCommandPayload.PayloadPtr))
THEN
  // add command.Distance.Y
  CreateCommandPayload.AddReal(_command.Distance.Y);
  // inc parameter counter
 _parameterCnt := _parameterCnt + 1;  
END_IF


// Check parameter must be added ? 
IF ( CheckAddParameter(CreateCommandPayload.PayloadPtr))
THEN
  // add command.Distance.Z
  CreateCommandPayload.AddReal(_command.Distance.Z);
  // inc parameter counter
 _parameterCnt := _parameterCnt + 1;  
END_IF


// Check parameter must be added ? 
IF ( CheckAddParameter(CreateCommandPayload.PayloadPtr))
THEN
  // add command.Distance.Rx
  CreateCommandPayload.AddReal(_command.Distance.Rx);
  // inc parameter counter
 _parameterCnt := _parameterCnt + 1;  
END_IF


// Check parameter must be added ? 
IF ( CheckAddParameter(CreateCommandPayload.PayloadPtr))
THEN
  // add command.Distance.Ry
  CreateCommandPayload.AddReal(_command.Distance.Ry);
  // inc parameter counter
 _parameterCnt := _parameterCnt + 1;  
END_IF


// Check parameter must be added ? 
IF ( CheckAddParameter(CreateCommandPayload.PayloadPtr))
THEN
  // add command.Distance.Rz
  CreateCommandPayload.AddReal(_command.Distance.Rz);
  // inc parameter counter
 _parameterCnt := _parameterCnt + 1;  
END_IF


// Check parameter must be added ? 
IF ( CheckAddParameter(CreateCommandPayload.PayloadPtr))
THEN
  // add command.Distance.Config
  CreateCommandPayload.AddArmConfig(_command.Distance.Config);
  // inc parameter counter
 _parameterCnt := _parameterCnt + 1;  
END_IF


// Check parameter must be added ? 
IF ( CheckAddParameter(CreateCommandPayload.PayloadPtr))
THEN
  // add command.Distance.TurnNumber
  CreateCommandPayload.AddTurnNumber(_command.Distance.TurnNumber);
  // inc parameter counter
 _parameterCnt := _parameterCnt + 1;  
END_IF


// Check parameter must be added ? 
IF ( CheckAddParameter(CreateCommandPayload.PayloadPtr))
THEN
  // add command.Distance.E1
  CreateCommandPayload.AddReal(_command.Distance.E1);
  // inc parameter counter
 _parameterCnt := _parameterCnt + 1;  
END_IF


// Check parameter must be added ? 
IF ( CheckAddParameter(CreateCommandPayload.PayloadPtr))
THEN
  // add command.Manipulation
  CreateCommandPayload.AddBool(_command.Manipulation);
  // inc parameter counter
 _parameterCnt := _parameterCnt + 1;  
END_IF


// Check parameter must be added ? 
IF ( CheckAddParameter(CreateCommandPayload.PayloadPtr))
THEN
  // add command.Reserve3
  CreateCommandPayload.AddByte(_command.Reserve3);
  // inc parameter counter
 _parameterCnt := _parameterCnt + 1;  
END_IF


// Check parameter must be added ? 
IF ( CheckAddParameter(CreateCommandPayload.PayloadPtr))
THEN
  // add command.ConfigMode[0]
  CreateCommandPayload.AddByte(_command.ConfigMode[0]);
  // inc parameter counter
 _parameterCnt := _parameterCnt + 1;  
END_IF


// Check parameter must be added ? 
IF ( CheckAddParameter(CreateCommandPayload.PayloadPtr))
THEN
  // add command.ConfigMode[1]
  CreateCommandPayload.AddByte(_command.ConfigMode[1]);
  // inc parameter counter
 _parameterCnt := _parameterCnt + 1;  
END_IF


// Check parameter must be added ? 
IF ( CheckAddParameter(CreateCommandPayload.PayloadPtr))
THEN
  // add command.ReferenceType
  CreateCommandPayload.AddUsint(_command.ReferenceType);
  // inc parameter counter
 _parameterCnt := _parameterCnt + 1;  
END_IF


// Check parameter must be added ? 
IF ( CheckAddParameter(CreateCommandPayload.PayloadPtr))
THEN
  // add command.TurnMode
  CreateCommandPayload.AddUsint(_command.TurnMode);
  // inc parameter counter
 _parameterCnt := _parameterCnt + 1;  
END_IF


// Check parameter must be added ? 
IF ( CheckAddParameter(CreateCommandPayload.PayloadPtr))
THEN
  // add command.MoveTime
  CreateCommandPayload.AddUint(_command.MoveTime);
  // inc parameter counter
 _parameterCnt := _parameterCnt + 1;  
END_IF


// Check parameter must be added ? 
IF ( CheckAddParameter(CreateCommandPayload.PayloadPtr))
THEN
  // add command.Distance.E2
  CreateCommandPayload.AddReal(_command.Distance.E2);
  // inc parameter counter
 _parameterCnt := _parameterCnt + 1;  
END_IF


// Check parameter must be added ? 
IF ( CheckAddParameter(CreateCommandPayload.PayloadPtr))
THEN
  // add command.Distance.E3
  CreateCommandPayload.AddReal(_command.Distance.E3);
  // inc parameter counter
 _parameterCnt := _parameterCnt + 1;  
END_IF


// Check parameter must be added ? 
IF ( CheckAddParameter(CreateCommandPayload.PayloadPtr))
THEN
  // add command.Distance.E4
  CreateCommandPayload.AddReal(_command.Distance.E4);
  // inc parameter counter
 _parameterCnt := _parameterCnt + 1;  
END_IF


// Check parameter must be added ? 
IF ( CheckAddParameter(CreateCommandPayload.PayloadPtr))
THEN
  // add command.Distance.E5
  CreateCommandPayload.AddReal(_command.Distance.E5);
  // inc parameter counter
 _parameterCnt := _parameterCnt + 1;  
END_IF


// Check parameter must be added ? 
IF ( CheckAddParameter(CreateCommandPayload.PayloadPtr))
THEN
  // add command.Distance.E6
  CreateCommandPayload.AddReal(_command.Distance.E6);
  // inc parameter counter
 _parameterCnt := _parameterCnt + 1;  
END_IF


// Create logging
CreateCommandPayloadLog(AxesGroup := AxesGroup, ParameterCnt := _parameterCnt);
                
END_METHOD

METHOD INTERNAL CreateCommandPayloadLog
VAR_IN_OUT
  /// Robot assignment of function
  AxesGroup : AxesGroup; 
END_VAR
VAR_INPUT
  /// Parameter count
  ParameterCnt : DINT;
END_VAR
VAR 
  /// internal index for loops
 _idx : DINT;
END_VAR
                  // Create log entry for Parameter start
CreateLogMessagePara1 ( Timestamp   := AxesGroup.State.SystemTime,
                        MessageType := MessageType.CMD,
                        Severity    := Severity.DEBUG,
                        MessageCode := 0,
                        MessageText := 'Create command payload with {1} parameter(s) :',
                        Para1       := DINT_TO_STRING(ParameterCnt));
  
// Create log entry for EmitterID[x]
FOR _idx := 0 TO 3
DO
  // Return if no parameter is remaining...
  IF ( ParameterCnt = 0 ) THEN RETURN; END_IF
  // dec remaining parameter(s)                        
  ParameterCnt := ParameterCnt - 1;
  // Create log entry for Command.EmitterID
  CreateLogMessagePara2 ( Timestamp   := AxesGroup.State.SystemTime,
                          MessageType := MessageType.CMD,
                          Severity    := Severity.DEBUG,
                          MessageCode := 0,
                          MessageText := 'Command.EmitterID[{2}] = {1}',
                          Para1       :=  SINT_TO_STRING(_command.EmitterID[_idx]),
                          Para2       :=  DINT_TO_STRING(_idx));
END_FOR


// Return if no parameter is remaining...
IF ( ParameterCnt = 0 ) THEN RETURN; END_IF
// dec remaining parameter(s)                        
ParameterCnt := ParameterCnt - 1;
// Create log entry for ListenerID
CreateLogMessagePara1 ( Timestamp   := AxesGroup.State.SystemTime,
                        MessageType := MessageType.CMD,
                        Severity    := Severity.DEBUG,
                        MessageCode := 0,
                        MessageText := 'Command.ListenerID = {1}',
                        Para1       :=  SINT_TO_STRING(_command.ListenerID));
                        

// Return if no parameter is remaining...
IF ( ParameterCnt = 0 ) THEN RETURN; END_IF
// dec remaining parameter(s)                        
ParameterCnt := ParameterCnt - 1;
// Create log entry for Reserve
CreateLogMessagePara1 ( Timestamp   := AxesGroup.State.SystemTime,
                        MessageType := MessageType.CMD,
                        Severity    := Severity.DEBUG,
                        MessageCode := 0,
                        MessageText := 'Command.Reserve = {1}',
                        Para1       :=  BYTE_TO_STRING(_command.Reserve));


// Return if no parameter is remaining...
IF ( ParameterCnt = 0 ) THEN RETURN; END_IF
// dec remaining parameter(s)                        
ParameterCnt := ParameterCnt - 1;
// Create log entry for VelocityRate
CreateLogMessagePara1 ( Timestamp   := AxesGroup.State.SystemTime,
                        MessageType := MessageType.CMD,
                        Severity    := Severity.DEBUG,
                        MessageCode := 0,
                        MessageText := 'Command.VelocityRate = {1}',
                        Para1       :=  UINT_TO_STRING(_command.VelocityRate));


// Return if no parameter is remaining...
IF ( ParameterCnt = 0 ) THEN RETURN; END_IF
// dec remaining parameter(s)                        
ParameterCnt := ParameterCnt - 1;
// Create log entry for AccelerationRate
CreateLogMessagePara1 ( Timestamp   := AxesGroup.State.SystemTime,
                        MessageType := MessageType.CMD,
                        Severity    := Severity.DEBUG,
                        MessageCode := 0,
                        MessageText := 'Command.AccelerationRate = {1}',
                        Para1       :=  UINT_TO_STRING(_command.AccelerationRate));
                        

// Return if no parameter is remaining...
IF ( ParameterCnt = 0 ) THEN RETURN; END_IF
// dec remaining parameter(s)                        
ParameterCnt := ParameterCnt - 1;
// Create log entry for DecelerationRate
CreateLogMessagePara1 ( Timestamp   := AxesGroup.State.SystemTime,
                        MessageType := MessageType.CMD,
                        Severity    := Severity.DEBUG,
                        MessageCode := 0,
                        MessageText := 'Command.DecelerationRate = {1}',
                        Para1       :=  UINT_TO_STRING(_command.DecelerationRate));


// Return if no parameter is remaining...
IF ( ParameterCnt = 0 ) THEN RETURN; END_IF
// dec remaining parameter(s)                        
ParameterCnt := ParameterCnt - 1;
// Create log entry for JerkRate
CreateLogMessagePara1 ( Timestamp   := AxesGroup.State.SystemTime,
                        MessageType := MessageType.CMD,
                        Severity    := Severity.DEBUG,
                        MessageCode := 0,
                        MessageText := 'Command.JerkRate = {1}',
                        Para1       :=  UINT_TO_STRING(_command.JerkRate));


// Return if no parameter is remaining...
IF ( ParameterCnt = 0 ) THEN RETURN; END_IF
// dec remaining parameter(s)                        
ParameterCnt := ParameterCnt - 1;
// Create log entry for ToolNo
CreateLogMessagePara1 ( Timestamp   := AxesGroup.State.SystemTime,
                        MessageType := MessageType.CMD,
                        Severity    := Severity.DEBUG,
                        MessageCode := 0,
                        MessageText := 'Command.ToolNo = {1}',
                        Para1       :=  USINT_TO_STRING(_command.ToolNo));


// Return if no parameter is remaining...
IF ( ParameterCnt = 0 ) THEN RETURN; END_IF
// dec remaining parameter(s)                        
ParameterCnt := ParameterCnt - 1;
// Create log entry for FrameNo
CreateLogMessagePara1 ( Timestamp   := AxesGroup.State.SystemTime,
                        MessageType := MessageType.CMD,
                        Severity    := Severity.DEBUG,
                        MessageCode := 0,
                        MessageText := 'Command.FrameNo = {1}',
                        Para1       :=  USINT_TO_STRING(_command.FrameNo));


// Return if no parameter is remaining...
IF ( ParameterCnt = 0 ) THEN RETURN; END_IF
// dec remaining parameter(s)                        
ParameterCnt := ParameterCnt - 1;
// Create log entry for BlendingMode
CreateLogMessagePara1 ( Timestamp   := AxesGroup.State.SystemTime,
                        MessageType := MessageType.CMD,
                        Severity    := Severity.DEBUG,
                        MessageCode := 0,
                        MessageText := 'Command.BlendingMode = {1}',
                        Para1       :=  BLENDING_MODE_TO_STRING(_command.BlendingMode));


// Return if no parameter is remaining...
IF ( ParameterCnt = 0 ) THEN RETURN; END_IF
// dec remaining parameter(s)                        
ParameterCnt := ParameterCnt - 1;
// Create log entry for Reserve
CreateLogMessagePara1 ( Timestamp   := AxesGroup.State.SystemTime,
                        MessageType := MessageType.CMD,
                        Severity    := Severity.DEBUG,
                        MessageCode := 0,
                        MessageText := 'Command.Reserve = {1}',
                        Para1       :=  BYTE_TO_STRING(_command.Reserve));


// Return if no parameter is remaining...
IF ( ParameterCnt = 0 ) THEN RETURN; END_IF
// dec remaining parameter(s)                        
ParameterCnt := ParameterCnt - 1;
// Create log entry for BlendingParameter[0]
CreateLogMessagePara1 ( Timestamp   := AxesGroup.State.SystemTime,
                        MessageType := MessageType.CMD,
                        Severity    := Severity.DEBUG,
                        MessageCode := 0,
                        MessageText := 'Command.BlendingParameter[0] = {1}',
                        Para1       :=  REAL_TO_STRING(_command.BlendingParameter[0]));


// Return if no parameter is remaining...
IF ( ParameterCnt = 0 ) THEN RETURN; END_IF
// dec remaining parameter(s)                        
ParameterCnt := ParameterCnt - 1;
// Create log entry for BlendingParameter[1]
CreateLogMessagePara1 ( Timestamp   := AxesGroup.State.SystemTime,
                        MessageType := MessageType.CMD,
                        Severity    := Severity.DEBUG,
                        MessageCode := 0,
                        MessageText := 'Command.BlendingParameter[1] = {1}',
                        Para1       :=  REAL_TO_STRING(_command.BlendingParameter[1]));


// Return if no parameter is remaining...
IF ( ParameterCnt = 0 ) THEN RETURN; END_IF
// dec remaining parameter(s)                        
ParameterCnt := ParameterCnt - 1;
// Create log entry for Distance.X
CreateLogMessagePara1 ( Timestamp   := AxesGroup.State.SystemTime,
                        MessageType := MessageType.CMD,
                        Severity    := Severity.DEBUG,
                        MessageCode := 0,
                        MessageText := 'Command.Distance.X = {1}',
                        Para1       :=  REAL_TO_STRING(_command.Distance.X));


// Return if no parameter is remaining...
IF ( ParameterCnt = 0 ) THEN RETURN; END_IF
// dec remaining parameter(s)                        
ParameterCnt := ParameterCnt - 1;
// Create log entry for Distance.Y
CreateLogMessagePara1 ( Timestamp   := AxesGroup.State.SystemTime,
                        MessageType := MessageType.CMD,
                        Severity    := Severity.DEBUG,
                        MessageCode := 0,
                        MessageText := 'Command.Distance.Y = {1}',
                        Para1       :=  REAL_TO_STRING(_command.Distance.Y));


// Return if no parameter is remaining...
IF ( ParameterCnt = 0 ) THEN RETURN; END_IF
// dec remaining parameter(s)                        
ParameterCnt := ParameterCnt - 1;
// Create log entry for Distance.Z
CreateLogMessagePara1 ( Timestamp   := AxesGroup.State.SystemTime,
                        MessageType := MessageType.CMD,
                        Severity    := Severity.DEBUG,
                        MessageCode := 0,
                        MessageText := 'Command.Distance.Z = {1}',
                        Para1       :=  REAL_TO_STRING(_command.Distance.Z));


// Return if no parameter is remaining...
IF ( ParameterCnt = 0 ) THEN RETURN; END_IF
// dec remaining parameter(s)                        
ParameterCnt := ParameterCnt - 1;
// Create log entry for Distance.Rx
CreateLogMessagePara1 ( Timestamp   := AxesGroup.State.SystemTime,
                        MessageType := MessageType.CMD,
                        Severity    := Severity.DEBUG,
                        MessageCode := 0,
                        MessageText := 'Command.Distance.Rx = {1}',
                        Para1       :=  REAL_TO_STRING(_command.Distance.Rx));


// Return if no parameter is remaining...
IF ( ParameterCnt = 0 ) THEN RETURN; END_IF
// dec remaining parameter(s)                        
ParameterCnt := ParameterCnt - 1;
// Create log entry for Distance.Ry
CreateLogMessagePara1 ( Timestamp   := AxesGroup.State.SystemTime,
                        MessageType := MessageType.CMD,
                        Severity    := Severity.DEBUG,
                        MessageCode := 0,
                        MessageText := 'Command.Distance.Ry = {1}',
                        Para1       :=  REAL_TO_STRING(_command.Distance.Ry));


// Return if no parameter is remaining...
IF ( ParameterCnt = 0 ) THEN RETURN; END_IF
// dec remaining parameter(s)                        
ParameterCnt := ParameterCnt - 1;
// Create log entry for Distance.Rz
CreateLogMessagePara1 ( Timestamp   := AxesGroup.State.SystemTime,
                        MessageType := MessageType.CMD,
                        Severity    := Severity.DEBUG,
                        MessageCode := 0,
                        MessageText := 'Command.Distance.Rz = {1}',
                        Para1       :=  REAL_TO_STRING(_command.Distance.Rz));


// Return if no parameter is remaining...
IF ( ParameterCnt = 0 ) THEN RETURN; END_IF
// dec remaining parameter(s)                        
ParameterCnt := ParameterCnt - 1;
// Create log entry for Distance.Config
CreateLogMessagePara1 ( Timestamp   := AxesGroup.State.SystemTime,
                        MessageType := MessageType.CMD,
                        Severity    := Severity.DEBUG,
                        MessageCode := 0,
                        MessageText := 'Command.Distance.Config = {1}',
                        Para1       :=  ARM_CONFIG_TO_STRING(_command.Distance.Config));


// Return if no parameter is remaining...
IF ( ParameterCnt = 0 ) THEN RETURN; END_IF
// dec remaining parameter(s)                        
ParameterCnt := ParameterCnt - 1;
// Create log entry for Distance.Reserve
CreateLogMessagePara1 ( Timestamp   := AxesGroup.State.SystemTime,
                        MessageType := MessageType.CMD,
                        Severity    := Severity.DEBUG,
                        MessageCode := 0,
                        MessageText := 'Command.Distance.Reserve = {1}',
                        Para1       :=  BYTE_TO_STRING(_command.Reserve));


// Return if no parameter is remaining...
IF ( ParameterCnt = 0 ) THEN RETURN; END_IF
// dec remaining parameter(s)                        
ParameterCnt := ParameterCnt - 1;
// Create log entry for Distance.TurnNumber[0]
CreateLogMessagePara1 ( Timestamp   := AxesGroup.State.SystemTime,
                        MessageType := MessageType.CMD,
                        Severity    := Severity.DEBUG,
                        MessageCode := 0,
                        MessageText := 'Command.Distance.TurnNumber[0] = {1}',
                        Para1       :=  BYTE_TO_STRING(CombineHalfSints(HalfSintHi := _command.Distance.TurnNumber.J2Turns,
                                                                        HalfSintLo := _command.Distance.TurnNumber.J1Turns)));


// Return if no parameter is remaining...
IF ( ParameterCnt = 0 ) THEN RETURN; END_IF
// dec remaining parameter(s)                        
ParameterCnt := ParameterCnt - 1;
// Create log entry for Distance.TurnNumber[1]
CreateLogMessagePara1 ( Timestamp   := AxesGroup.State.SystemTime,
                        MessageType := MessageType.CMD,
                        Severity    := Severity.DEBUG,
                        MessageCode := 0,
                        MessageText := 'Command.Distance.TurnNumber[1] = {1}',
                        Para1       :=  BYTE_TO_STRING(CombineHalfSints(HalfSintHi := _command.Distance.TurnNumber.J4Turns, 
                                                                        HalfSintLo := _command.Distance.TurnNumber.J3Turns)));


// Return if no parameter is remaining...
IF ( ParameterCnt = 0 ) THEN RETURN; END_IF
// dec remaining parameter(s)                        
ParameterCnt := ParameterCnt - 1;
// Create log entry for Distance.TurnNumber[2]
CreateLogMessagePara1 ( Timestamp   := AxesGroup.State.SystemTime,
                        MessageType := MessageType.CMD,
                        Severity    := Severity.DEBUG,
                        MessageCode := 0,
                        MessageText := 'Command.ReferencePosition.TurnNumber[2] = {1}',
                        Para1       :=  BYTE_TO_STRING(CombineHalfSints(HalfSintHi := _command.Distance.TurnNumber.J6Turns, 
                                                                        HalfSintLo := _command.Distance.TurnNumber.J5Turns)));


// Return if no parameter is remaining...
IF ( ParameterCnt = 0 ) THEN RETURN; END_IF
// dec remaining parameter(s)                        
ParameterCnt := ParameterCnt - 1;
// Create log entry for Distance.TurnNumber[3]
CreateLogMessagePara1 ( Timestamp   := AxesGroup.State.SystemTime,
                        MessageType := MessageType.CMD,
                        Severity    := Severity.DEBUG,
                        MessageCode := 0,
                        MessageText := 'Command.Distance.TurnNumber[3] = {1}',
                        Para1       :=  SINT_TO_STRING(_command.Distance.TurnNumber.E1Turns));


// Return if no parameter is remaining...
IF ( ParameterCnt = 0 ) THEN RETURN; END_IF
// dec remaining parameter(s)                        
ParameterCnt := ParameterCnt - 1;
// Create log entry for Distance.E1
CreateLogMessagePara1 ( Timestamp   := AxesGroup.State.SystemTime,
                        MessageType := MessageType.CMD,
                        Severity    := Severity.DEBUG,
                        MessageCode := 0,
                        MessageText := 'Command.Distance.E1 = {1}',
                        Para1       :=  REAL_TO_STRING(_command.Distance.E1));


// Return if no parameter is remaining...
IF ( ParameterCnt = 0 ) THEN RETURN; END_IF
// dec remaining parameter(s)                        
ParameterCnt := ParameterCnt - 1;
// Create log entry for Manipulation
CreateLogMessagePara1 ( Timestamp   := AxesGroup.State.SystemTime,
                        MessageType := MessageType.CMD,
                        Severity    := Severity.DEBUG,
                        MessageCode := 0,
                        MessageText := 'Command.Manipulation = {1}',
                        Para1       :=  BOOL_TO_STRING(_command.Manipulation));


// Return if no parameter is remaining...
IF ( ParameterCnt = 0 ) THEN RETURN; END_IF
// dec remaining parameter(s)                        
ParameterCnt := ParameterCnt - 1;
// Create log entry for Reserve
CreateLogMessagePara1 ( Timestamp   := AxesGroup.State.SystemTime,
                        MessageType := MessageType.CMD,
                        Severity    := Severity.DEBUG,
                        MessageCode := 0,
                        MessageText := 'Command.Reserve = {1}',
                        Para1       :=  BYTE_TO_STRING(_command.Reserve));


// Return if no parameter is remaining...
IF ( ParameterCnt = 0 ) THEN RETURN; END_IF
// dec remaining parameter(s)                        
ParameterCnt := ParameterCnt - 1;
// Create log entry for ConfigMode[0]
CreateLogMessagePara1 ( Timestamp   := AxesGroup.State.SystemTime,
                        MessageType := MessageType.CMD,
                        Severity    := Severity.DEBUG,
                        MessageCode := 0,
                        MessageText := 'Command.ConfigMode[0] = {1}',
                        Para1       :=  BYTE_TO_STRING_BIN(_command.ConfigMode[0]));


// Return if no parameter is remaining...
IF ( ParameterCnt = 0 ) THEN RETURN; END_IF
// dec remaining parameter(s)                        
ParameterCnt := ParameterCnt - 1;
// Create log entry for ConfigMode[1]
CreateLogMessagePara1 ( Timestamp   := AxesGroup.State.SystemTime,
                        MessageType := MessageType.CMD,
                        Severity    := Severity.DEBUG,
                        MessageCode := 0,
                        MessageText := 'Command.ConfigMode[1] = {1}',
                        Para1       :=  BYTE_TO_STRING_BIN(_command.ConfigMode[1]));


// Return if no parameter is remaining...
IF ( ParameterCnt = 0 ) THEN RETURN; END_IF
// dec remaining parameter(s)                        
ParameterCnt := ParameterCnt - 1;
// Create log entry for ReferenceType
CreateLogMessagePara1 ( Timestamp   := AxesGroup.State.SystemTime,
                        MessageType := MessageType.CMD,
                        Severity    := Severity.DEBUG,
                        MessageCode := 0,
                        MessageText := 'Command.ReferenceType = {1}',
                        Para1       :=  REFERENCE_TYPE_TO_STRING(_command.ReferenceType));


// Return if no parameter is remaining...
IF ( ParameterCnt = 0 ) THEN RETURN; END_IF
// dec remaining parameter(s)                        
ParameterCnt := ParameterCnt - 1;
// Create log entry for TurnMode
CreateLogMessagePara1 ( Timestamp   := AxesGroup.State.SystemTime,
                        MessageType := MessageType.CMD,
                        Severity    := Severity.DEBUG,
                        MessageCode := 0,
                        MessageText := 'Command.TurnMode = {1}',
                        Para1       :=  TURN_MODE_TO_STRING(_command.TurnMode));


// Return if no parameter is remaining...
IF ( ParameterCnt = 0 ) THEN RETURN; END_IF
// dec remaining parameter(s)                        
ParameterCnt := ParameterCnt - 1;
// Create log entry for MoveTime
CreateLogMessagePara1 ( Timestamp   := AxesGroup.State.SystemTime,
                        MessageType := MessageType.CMD,
                        Severity    := Severity.DEBUG,
                        MessageCode := 0,
                        MessageText := 'Command.MoveTime = {1}',
                        Para1       :=  UINT_TO_STRING(_command.MoveTime));


// Return if no parameter is remaining...
IF ( ParameterCnt = 0 ) THEN RETURN; END_IF
// dec remaining parameter(s)                        
ParameterCnt := ParameterCnt - 1;
// Create log entry for Distance.E2
CreateLogMessagePara1 ( Timestamp   := AxesGroup.State.SystemTime,
                        MessageType := MessageType.CMD,
                        Severity    := Severity.DEBUG,
                        MessageCode := 0,
                        MessageText := 'Command.Distance.E2 = {1}',
                        Para1       :=  REAL_TO_STRING(_command.Distance.E2));


// Return if no parameter is remaining...
IF ( ParameterCnt = 0 ) THEN RETURN; END_IF
// dec remaining parameter(s)                        
ParameterCnt := ParameterCnt - 1;
// Create log entry for Distance.E3
CreateLogMessagePara1 ( Timestamp   := AxesGroup.State.SystemTime,
                        MessageType := MessageType.CMD,
                        Severity    := Severity.DEBUG,
                        MessageCode := 0,
                        MessageText := 'Command.Distance.E3 = {1}',
                        Para1       :=  REAL_TO_STRING(_command.Distance.E3));


// Return if no parameter is remaining...
IF ( ParameterCnt = 0 ) THEN RETURN; END_IF
// dec remaining parameter(s)                        
ParameterCnt := ParameterCnt - 1;
// Create log entry for Distance.E4
CreateLogMessagePara1 ( Timestamp   := AxesGroup.State.SystemTime,
                        MessageType := MessageType.CMD,
                        Severity    := Severity.DEBUG,
                        MessageCode := 0,
                        MessageText := 'Command.Distance.E4 = {1}',
                        Para1       :=  REAL_TO_STRING(_command.Distance.E4));


// Return if no parameter is remaining...
IF ( ParameterCnt = 0 ) THEN RETURN; END_IF
// dec remaining parameter(s)                        
ParameterCnt := ParameterCnt - 1;
// Create log entry for Distance.E5
CreateLogMessagePara1 ( Timestamp   := AxesGroup.State.SystemTime,
                        MessageType := MessageType.CMD,
                        Severity    := Severity.DEBUG,
                        MessageCode := 0,
                        MessageText := 'Command.Distance.E5 = {1}',
                        Para1       :=  REAL_TO_STRING(_command.Distance.E5));


// Return if no parameter is remaining...
IF ( ParameterCnt = 0 ) THEN RETURN; END_IF
// dec remaining parameter(s)                        
ParameterCnt := ParameterCnt - 1;
// Create log entry for Distance.E6
CreateLogMessagePara1 ( Timestamp   := AxesGroup.State.SystemTime,
                        MessageType := MessageType.CMD,
                        Severity    := Severity.DEBUG,
                        MessageCode := 0,
                        MessageText := 'Command.Distance.E6 = {1}',
                        Para1       :=  REAL_TO_STRING(_command.Distance.E6));

                
END_METHOD

METHOD FB_init : BOOL
VAR_INPUT
  /// if TRUE, the retain variables are initialized (warm start / cold start)
  bInitRetains : BOOL; 
  /// if TRUE, the instance afterwards gets moved into the copy code (online change)
  bInCopyCode  : BOOL;  
END_VAR
                  MyType := 'MC_MoveDirectRelativeFB';

ExecMode     := ExecutionMode.SEQUENCE_PRIMARY;
Priority     := PriorityLevel.NORMAL;
AbortingMode := AbortingModeEnum.BUFFER;  
SequenceFlag := SequenceFlagEnum.PRIMARY_SEQUENCE;  

                
END_METHOD

METHOD PROTECTED OnApplyOutCmd
VAR_INPUT
  /// Command message state
  State : CmdMessageState;
END_VAR
                  IF ( State = CmdMessageState.EMPTY ) 
THEN
  // Reset command outputs
  SysDepMemSet(pDest := ADR(OutCmd), Value := 0, DataLen := SIZEOF(OutCmd));         
END_IF

IF (( State = CmdMessageState.ACTIVE ) OR
    ( State = CmdMessageState.DONE   ))
THEN
  // Update results
  OutCmd.Progress          :=  PERCENT_UINT_TO_REAL( Value := _response.Progress, IsOptional := TRUE);
  OutCmd.FollowID          := _response.OriginID;
  OutCmd.RemainingDistance := _response.RemainingDistance;
END_IF
                
END_METHOD

METHOD PROTECTED OnExecRun : DINT
VAR_IN_OUT
  /// Robot assignment of function
  AxesGroup : AxesGroup; 
END_VAR
                  // call base implementation
SUPER^.OnExecRun(AxesGroup := AxesGroup);

CASE _stepCmd OF
  
  00:  IF ( _execute_R.Q ) AND ( NOT Error) 
       THEN
         // Check function is supported and parameter are valid ?
         IF (( CheckFunctionSupported( AxesGroup := AxesGroup )) AND
             ( CheckParameterValid   ( AxesGroup := AxesGroup )))      
         THEN
           // set busy flag
           Busy := TRUE;
           // Reset command outputs
           SysDepMemSet(pDest := ADR(OutCmd), Value := 0, DataLen := SIZEOF(OutCmd));         
           // apply command parameter
          _parCmd := ParCmd;
           // init parameter sequence
          _command.ParSeq := 1;
           // create command data
           CommandData := CreateCommandPayload(AxesGroup := AxesGroup);
           // Add command to active command register
          _uniqueID := AxesGroup.Acyclic.ActiveCommandRegister.AddCmd( pCommandFB := ADR(THIS^ ));     
           // set timeout
           SetTimeout(PT := _timeoutCmd, rTimer := _timerCmd);
           // inc step counter
          _stepCmd := _stepCmd + 1;
         END_IF 
       END_IF
     

  01:  // Wait for responce received
       IF ( _responseReceived )
       THEN
         // reset response received flag
        _responseReceived := FALSE;
         // update state flags
         OnUpdateStateFlags(_response.State);
         // update state flags
         OnApplyOutCmd(_response.State);
        
         // Done, Aborted or Error ?
         IF (_response.State >= CmdMessageState.DONE )
         THEN
           // set timeout
           SetTimeout(PT := _timeoutCmd, rTimer := _timerCmd);
           // inc step counter
          _stepCmd := _stepCmd + 1; 
         END_IF
       END_IF
       

  02: IF ( NOT Execute)
      THEN
        Reset();  
      END_IF     
ELSE
  // invalid step
  SetError( ErrorID := RobotLibraryErrorIdEnum.ERR_INVALID_STEP, Overwrite := TRUE );
END_CASE


// Reset FB
IF ( NOT Execute )
THEN
  Reset();  
END_IF
                
END_METHOD

METHOD PROTECTED OnUpdateStateFlags
VAR_INPUT
  /// Command message state
  State : CmdMessageState;
END_VAR
                  // Reset State flags
Active             := FALSE;
CommandAborted     := FALSE;
CommandInterrupted := FALSE;
Done               := FALSE;

CASE State OF

  // No operation or process is active
  CmdMessageState.EMPTY               :;
  // Created but not yet started
  CmdMessageState.CREATED             :;
  // Buffered and awaiting execution
  CmdMessageState.BUFFERED            : CommandBuffered    := TRUE;
  // Buffered in planner for future execution
  CmdMessageState.BUFFERED_IN_PLANNER : CommandBuffered    := TRUE;
  // Currently active and in progress
  CmdMessageState.ACTIVE              : Active             := TRUE; 
  // Interrupted and awaiting continuation
  CmdMessageState.INTERRUPTED         : CommandInterrupted := TRUE;  
  // Requested for abort
  CmdMessageState.ABORT_REQUEST       :;
  // Successfully completed
  CmdMessageState.DONE                : Done               := TRUE;
                                        Busy               := FALSE;
  // Aborted before completion
  CmdMessageState.ABORTED             : CommandAborted     := TRUE;
                                        Busy               := FALSE;
  // Encountered an error during execution
  CmdMessageState.ERROR               : Error              := TRUE;
                                        Busy               := FALSE;
END_CASE
                
END_METHOD

METHOD INTERNAL ParseResponsePayload : DINT
VAR_INPUT
  /// Response data
  ResponseData : RobotLibraryResponseDataFB;
  /// Timestamp
  Timestamp    : SystemTime;  
END_VAR
VAR
  /// Parameter count
 _parameterCnt : DINT;
END_VAR
// Table 6-298: Received CMD payload (RC to PLC) of "MoveDirectRelative"
// --------------------------
// Header
// --------------------------
// Byte 00 : USINT   - ParSeq | State     
// Byte 01 : SINT    - AlarmMessageSeverity    
// Byte 02 : UINT    - AlarmMessageCode HB
// Byte 03 :         - AlarmMessageCode LB
// --------------------------
// Datablock
// --------------------------
// Byte 04 : USINT      - InvocationCounter
// Byte 05 : SINT       - Reserved
// Byte 06 : INT        - OriginID HW HB
// Byte 07 :            - OriginID HW LB
// Byte 08 : UINT       - Progress HW HB
// Byte 09 :            - Progress HW LB
// Byte 10 : REAL       - RemainingDistance HW HB
// Byte 11 :            - RemainingDistance HW LB
// Byte 12 :            - RemainingDistance LW HB
// Byte 13 :            - RemainingDistance LW LB
                  // call base implementation to parse the header from payload buffer
ResponseData.PayloadPtr := SUPER^.ParseResponsePayload(ResponseData := ResponseData, Timestamp := Timestamp);

// copy parsed header to response
_response.ParSeq               := _rspHeader.ParSeq;
_response.State                := _rspHeader.State;
_response.AlarmMessageSeverity := _rspHeader.AlarmMessageSeverity;
_response.AlarmMessageCode     := _rspHeader.AlarmMessageCode;


// Check payload remaining ? 
IF ( ResponseData.IsPayloadRemaining)
THEN
  // Get Response.InvocationCounter
 _response.InvocationCounter := ResponseData.GetUsint();
  // inc parameter counter
 _parameterCnt := _parameterCnt + 1;
END_IF


// Check payload remaining ? 
IF ( ResponseData.IsPayloadRemaining)
THEN
  // Get Response.Reserve
 _response.Reserve := ResponseData.GetSint();
  // inc parameter counter
 _parameterCnt := _parameterCnt + 1;
END_IF


// Check payload remaining ? 
IF ( ResponseData.IsPayloadRemaining)
THEN
  // Get Response.OriginID
 _response.OriginID := ResponseData.GetInt();
  // inc parameter counter
 _parameterCnt := _parameterCnt + 1;
END_IF


// Check payload remaining ? 
IF ( ResponseData.IsPayloadRemaining)
THEN
  // Get Response.Progress
 _response.Progress := ResponseData.GetUint();
  // inc parameter counter
 _parameterCnt := _parameterCnt + 1;
END_IF


// Check payload remaining ? 
IF ( ResponseData.IsPayloadRemaining)
THEN
  // Get Response.RemainingDistance
 _response.RemainingDistance := ResponseData.GetReal();
  // inc parameter counter
 _parameterCnt := _parameterCnt + 1;
END_IF

 
// Create logging
ParseResponsePayloadLog(ResponseData := ResponseData, Timestamp := Timestamp, ParameterCnt := _parameterCnt);
                
END_METHOD

METHOD INTERNAL ParseResponsePayloadLog
VAR_INPUT
  /// Response data
  ResponseData : RobotLibraryResponseDataFB;
  /// Timestamp
  Timestamp    : SystemTime;  
  /// Parameter count
  ParameterCnt : DINT;
END_VAR
                  // Create log entry for Parameter start
CreateLogMessagePara1 ( Timestamp   := Timestamp,
                        MessageType := MessageType.CMD,
                        Severity    := Severity.DEBUG,
                        MessageCode := 0,
                        MessageText := '{1} parameter(s) to parse from the response data:',
                        Para1       := DINT_TO_STRING(ParameterCnt));
                        

// Return if no parameter is remaining...
IF ( ParameterCnt = 0 ) THEN RETURN; END_IF
// dec remaining parameter(s)                        
ParameterCnt := ParameterCnt - 1;
// Create log entry for InvocationCounter
CreateLogMessagePara1 ( Timestamp   := Timestamp,
                        MessageType := MessageType.CMD,
                        Severity    := Severity.DEBUG,
                        MessageCode := 0,
                        MessageText := 'Response.InvocationCounter = {1}',
                        Para1       :=  USINT_TO_STRING(_response.InvocationCounter));


// Return if no parameter is remaining...
IF ( ParameterCnt = 0 ) THEN RETURN; END_IF
// dec remaining parameter(s)                        
ParameterCnt := ParameterCnt - 1;
// Create log entry for Reserve
CreateLogMessagePara1 ( Timestamp   := Timestamp,
                        MessageType := MessageType.CMD,
                        Severity    := Severity.DEBUG,
                        MessageCode := 0,
                        MessageText := 'Response.Reserve = {1}',
                        Para1       :=  SINT_TO_STRING(_response.Reserve));


// Return if no parameter is remaining...
IF ( ParameterCnt = 0 ) THEN RETURN; END_IF
// dec remaining parameter(s)                        
ParameterCnt := ParameterCnt - 1;
// Create log entry for OriginID
CreateLogMessagePara1 ( Timestamp   := Timestamp,
                        MessageType := MessageType.CMD,
                        Severity    := Severity.DEBUG,
                        MessageCode := 0,
                        MessageText := 'Response.OriginID = {1}',
                        Para1       :=  INT_TO_STRING(_response.OriginID));


// Return if no parameter is remaining...
IF ( ParameterCnt = 0 ) THEN RETURN; END_IF
// dec remaining parameter(s)                        
ParameterCnt := ParameterCnt - 1;
// Create log entry for Progress
CreateLogMessagePara1 ( Timestamp   := Timestamp,
                        MessageType := MessageType.CMD,
                        Severity    := Severity.DEBUG,
                        MessageCode := 0,
                        MessageText := 'Response.Progress = {1}',
                        Para1       :=  UINT_TO_STRING(_response.Progress));


// Return if no parameter is remaining...
IF ( ParameterCnt = 0 ) THEN RETURN; END_IF
// dec remaining parameter(s)                        
ParameterCnt := ParameterCnt - 1;
// Create log entry for RemainingDistance
CreateLogMessagePara1 ( Timestamp   := Timestamp,
                        MessageType := MessageType.CMD,
                        Severity    := Severity.DEBUG,
                        MessageCode := 0,
                        MessageText := 'Response.RemainingDistance = {1}',
                        Para1       :=  REAL_TO_STRING(_response.RemainingDistance));
                
END_METHOD

METHOD PROTECTED Reset : DINT
VAR_INPUT
END_VAR
                  Reset := SUPER^.Reset();

Done               := FALSE;
Busy               := FALSE;
Active             := FALSE;
CommandBuffered    := FALSE;
CommandAborted     := FALSE;
CommandInterrupted := FALSE;

                
END_METHOD
END_FUNCTION_BLOCK

/// Move TCP to an absolute joint position (linear interpolation)
FUNCTION_BLOCK MC_MoveLinearAbsoluteJFB EXTENDS RobotLibraryBaseExecuteFB
// ------------------------------------------------------------------------- 
//  SRCI Robot Library                                                
// ------------------------------------------------------------------------- 
//                                                                           
//  Object:      MoveLinearAbsoluteJFB                                       
//  Author:      Thorsten Brach                                                
//  Date:        2024-06-01
//
//  Description:                                              
//   
//                                                                           
//  Copyright: 
//    (C) 2024 Thorsten Brach. All rights reserved                                                                                                                                            
//             Licensed under the MIT License.
//                                                                           
//  Disclaimer:                                                                           
//    This project is provided without any guarantee and can be used for   
//    private and commercial purposes. Any use is at the user’s 
//    own risk and responsibility.
//
// -------------------------------------------------------------------------
VAR_INPUT
  /// Parameter which determines the behavior towards the previously sent and still active or buffered commands
  AbortingMode       : AbortingMode;
  /// Defines the target sequence in which the command will be executed
  SequenceFlag       : SequenceFlag;
  /// command parameter
  ParCmd             : MoveLinearAbsoluteJParCmd;       
END_VAR

VAR_OUTPUT
  /// Command is transferred and confirmed by the RC
  CommandBuffered    : BOOL;
  /// The command takes control of the motion of the according axis group
  Active             : BOOL;
  /// The command was aborted by another command.
  CommandAborted     : BOOL;
  /// TRUE, while command is interrupted during execution and can be continued
  CommandInterrupted : BOOL;
  /// command outputs
  OutCmd             : MoveLinearAbsoluteJOutCmd;       
END_VAR

VAR
  /// internal copy of command parameter 
 _parCmd             : MoveLinearAbsoluteJParCmd;
  /// command data to send
 _command            : MoveLinearAbsoluteJSendData;
  /// response data received
 _response           : MoveLinearAbsoluteJRecvData;      
END_VAR

            SUPER^(AxesGroup := AxesGroup);
          

METHOD INTERNAL CheckAddParameter : BOOL
VAR_INPUT
  /// Payload pointer
  PayloadPtr : UDINT;
END_VAR
VAR
  /// Payload as byte array
  Payload    : ARRAY [1..SIZEOF(_command)] OF BYTE;
  /// Null Byte array 
  Null       : ARRAY [1..SIZEOF(_command)] OF BYTE;
  /// Data length to compare
  DataLen    : UDINT;
END_VAR
                  // Payload pointer must be decreased by one byte, because ADR(Payload) is already one byte !
PayloadPtr := LIMIT (0, PayloadPtr - 1, SIZEOF(Payload) -1);
// Convert command struct to payload array
SysDepMemCpy( pDest := ADR(Payload), pSrc := ADR(_command), DataLen := SIZEOF(_command));
// Calculate the data length to compare - at least one byte must be compared !
DataLen := LIMIT(1, SIZEOF(Payload) - PayloadPtr, SIZEOF(Payload)); 
// Compare Payload-Array with Null-Byte-Array
CheckAddParameter := SysDepMemCmp( pData1 := ADR(Payload) + PayloadPtr , pData2 := ADR(Null), DataLen := DataLen) <>  RobotLibraryConstants.OK ;
                
END_METHOD

METHOD PROTECTED CheckFunctionSupported : BOOL
VAR_IN_OUT
  /// Robot assignment of function
  AxesGroup : AxesGroup; 
END_VAR
                  CheckFunctionSupported := AxesGroup.State.RobotData.RCSupportedFunctions.MoveLinearAbsoluteJ;

IF ( NOT CheckFunctionSupported )
THEN
  // call base implementation for set error and create log entry
  SUPER^.CheckFunctionSupported(AxesGroup := AxesGroup);
END_IF
                
END_METHOD

METHOD PROTECTED CheckParameterChanged : BOOL
VAR_IN_OUT
  /// Robot assignment of function
  AxesGroup    : AxesGroup; 
END_VAR
                  // Check ParCmd Size is > 0, because MemCmp does not work correctly with size = 0
IF (SIZEOF(ParCmd) = 0) OR (_stepCmd = 0)
THEN 
  RETURN;
END_IF

// compare memory 
_parameterChanged := ( SysDepMemCmp(pData1 := ADR(ParCmd), pData2 := ADR(_parCmd), DataLen := SIZEOF(ParCmd)) <> RobotLibraryConstants.OK );

// check parameter valid ?
_parameterValid   := CheckParameterValid( AxesGroup := AxesGroup );

IF ((  _parameterChanged        )  AND 
    (  _parameterValid          )) OR
    (  _parameterUpdateInternal )  
THEN  
  // Create log entry for parameter changed event
  CreateLogMessagePara1 ( Timestamp   := AxesGroup.State.SystemTime,
                          MessageType := MessageType.CMD,
                          Severity    := Severity.DEBUG,
                          MessageCode := 0,
                          MessageText := 'NotifyParameterChanged Event {1}',
                          Para1       :=  '' );

  // reset internal flag for send parameter update
 _parameterUpdateInternal := FALSE;
  // update internal copy of parameters 
 _parCmd := ParCmd;
  // inc parameter sequence
 _command.ParSeq := _command.ParSeq + 1;
  // update command data  
  CommandData := CreateCommandPayload(AxesGroup := AxesGroup); // ( Access via reference to rCommandFB in ACR )
  // notify active command register 
  AxesGroup.Acyclic.ActiveCommandRegister.NotifyParameterChanged := _uniqueID;
END_IF
                
END_METHOD

METHOD PROTECTED CheckParameterValid : BOOL
VAR_IN_OUT
  /// Robot assignment of function
  AxesGroup : AxesGroup; 
END_VAR
VAR
  /// internal index for loops
 _idx : DINT;
END_VAR
                  CheckParameterValid := TRUE;

// Check AbortingMode valid ? 
IF (( AbortingMode <> AbortingModeEnum.BUFFER ) AND
    ( AbortingMode <> AbortingModeEnum.ABORT  ))  
THEN
  // Parameter not valid
  CheckParameterValid := FALSE;
  // Set error
  SetError( ErrorID := RobotLibraryErrorIdEnum.ERR_ABORTINGMODE_INVALID, Overwrite := TRUE );
  // Create log entry
  CreateLogMessagePara1 ( Timestamp   := AxesGroup.State.SystemTime,
                          MessageType := MessageType.CMD,
                          Severity    := Severity.ERROR,
                          MessageCode := ErrorID,
                          MessageText := 'Invalid Parameter AbortingMode = {1}',
                          Para1       := ABORTING_MODE_TO_STRING(AbortingMode));
  RETURN;                          
END_IF


// Check SequenceFlag valid ? 
IF (( SequenceFlag <> SequenceFlagEnum.PRIMARY_SEQUENCE   ) AND
    ( SequenceFlag <> SequenceFlagEnum.SECONDARY_SEQUENCE ))
THEN
  // Parameter not valid
  CheckParameterValid := FALSE;
  // Set error
  SetError( ErrorID := RobotLibraryErrorIdEnum.ERR_SEQFLAG_NOT_ALLOWED, Overwrite := TRUE );
  // Create log entry
  CreateLogMessagePara1 ( Timestamp   := AxesGroup.State.SystemTime,
                          MessageType := MessageType.CMD,
                          Severity    := Severity.ERROR,
                          MessageCode := ErrorID,
                          MessageText := 'Invalid Parameter SequenceFlag = {1}',
                          Para1       := SEQUENCE_FLAG_TO_STRING(SequenceFlag));
  RETURN;                          
END_IF


// Check ParCmd.JointPosition.J1 valid ? 
IF ( SysDepIsValidReal(ParCmd.JointPosition.J1) = FALSE ) 
THEN
  // Parameter not valid
  CheckParameterValid := FALSE;
  // Set error
  SetError( ErrorID := RobotLibraryErrorIdEnum.ERR_INVALID_PAR_CMD, Overwrite := TRUE );
  
  // Create log entry
  CreateLogMessagePara1 ( Timestamp   := AxesGroup.State.SystemTime,
                          MessageType := MessageType.CMD,
                          Severity    := Severity.ERROR,
                          MessageCode := ErrorID,
                          MessageText := 'Invalid Parameter ParCmd.JointPosition.J1 = {1}',
                          Para1       := VALID_REAL_TO_STRING(ParCmd.JointPosition.J1));
  RETURN;                          
END_IF


// Check ParCmd.JointPosition.J2 valid ? 
IF ( SysDepIsValidReal(ParCmd.JointPosition.J2) = FALSE ) 
THEN
  // Parameter not valid
  CheckParameterValid := FALSE;
  // Set error
  SetError( ErrorID := RobotLibraryErrorIdEnum.ERR_INVALID_PAR_CMD, Overwrite := TRUE );
  
  // Create log entry
  CreateLogMessagePara1 ( Timestamp   := AxesGroup.State.SystemTime,
                          MessageType := MessageType.CMD,
                          Severity    := Severity.ERROR,
                          MessageCode := ErrorID,
                          MessageText := 'Invalid Parameter ParCmd.JointPosition.J2 = {1}',
                          Para1       := VALID_REAL_TO_STRING(ParCmd.JointPosition.J2));
  RETURN;                          
END_IF


// Check ParCmd.JointPosition.J3 valid ? 
IF ( SysDepIsValidReal(ParCmd.JointPosition.J3) = FALSE ) 
THEN
  // Parameter not valid
  CheckParameterValid := FALSE;
  // Set error
  SetError( ErrorID := RobotLibraryErrorIdEnum.ERR_INVALID_PAR_CMD, Overwrite := TRUE );
  
  // Create log entry
  CreateLogMessagePara1 ( Timestamp   := AxesGroup.State.SystemTime,
                          MessageType := MessageType.CMD,
                          Severity    := Severity.ERROR,
                          MessageCode := ErrorID,
                          MessageText := 'Invalid Parameter ParCmd.JointPosition.J3 = {1}',
                          Para1       := VALID_REAL_TO_STRING(ParCmd.JointPosition.J3));
  RETURN;                          
END_IF


// Check ParCmd.JointPosition.J4 valid ? 
IF ( SysDepIsValidReal(ParCmd.JointPosition.J4) = FALSE ) 
THEN
  // Parameter not valid
  CheckParameterValid := FALSE;
  // Set error
  SetError( ErrorID := RobotLibraryErrorIdEnum.ERR_INVALID_PAR_CMD, Overwrite := TRUE );
  
